# B&R Automation Studio project acopos6d_issues (part 3)

#### brdkSTR.fun
```iecst
FUNCTION brdkStrAppendUdintToA : DINT (*Appends an UDINT to the end of a string. $RETURN=length;Length of the string.*) (*$GROUP=User,$CAT=User,$GROUPICON=User.png,$CATICON=User.png*)
	VAR_INPUT
		value : UDINT; (*UDINT value to be converted.*)
		pString : UDINT; (*String pointer to source string.*)
		base : USINT; (*0,10 = decimal, 2 = binary, 16 = hex.*)
		position : DINT; (*Append position. Negative numbers will count from end of string.*)
	END_VAR
END_FUNCTION

FUNCTION brdkStrAToDint : DINT (*Converts a string to a DINT type. $RETURN=value;DINT value.*) (*$GROUP=User,$CAT=User,$GROUPICON=User.png,$CATICON=User.png*)
	VAR_INPUT
		pString : UDINT; (*String pointer to source string.*)
		base : USINT; (*0,10 = decimal, 2 = binary, 16 = hex.*)
	END_VAR
END_FUNCTION

FUNCTION brdkStrAToDTStructure : DINT (*Converts a STRING of format yyyy-mm-dd hh:mm:ss.ms into a DTStructure. $RETURN=length;Length of the string.*) (*$GROUP=User,$CAT=User,$GROUPICON=User.png,$CATICON=User.png*)
	VAR_INPUT
		pString : UDINT; (*String pointer to source string.*)
		pDTStructure : UDINT; (*Pointer to the DTStructure.*)
	END_VAR
END_FUNCTION

FUNCTION brdkStrAToUdint : UDINT (*Converts a string to an UDINT type. $RETURN=value;UDINT value.*) (*$GROUP=User,$CAT=User,$GROUPICON=User.png,$CATICON=User.png*)
	VAR_INPUT
		pString : UDINT; (*String pointer to source string.*)
		base : USINT; (*0,10 = decimal, 2 = binary, 16 = hex.*)
	END_VAR
END_FUNCTION

FUNCTION brdkStrCat : UDINT (*Appends a copy of the source string to the end of the destination string. $RETURN=address;Address after the string.*) (*$GROUP=User,$CAT=User,$GROUPICON=User.png,$CATICON=User.png*)
	VAR_INPUT
		pDestination : UDINT; (*Destination string pointer.*)
		pSource : UDINT; (*Source string pointer.*)
	END_VAR
END_FUNCTION

FUNCTION brdkStrCatAtChar : DINT (*Appends a copy of the source string to the char position of the destination string. $RETURN=index;Index in destination string where the source string is appended. -1 if char is not found.*) (*$GROUP=User,$CAT=User,$GROUPICON=User.png,$CATICON=User.png*)
	VAR_INPUT
		pDestination : UDINT; (*Destination string pointer.*)
		pSource : UDINT; (*Source string pointer.*)
		pChar : UDINT; (*Char pointer.*)
		direction : DINT; (*0 = first appearance of char, -1 = last appearance of char.*)
		greedy : BOOL; (*If true the source string is appended to the char position. If false the char is still present in the destination string.*)
	END_VAR
END_FUNCTION

FUNCTION brdkStrCharAt : USINT (*Returns the character at the specified index. $RETURN=coding;ASCII coding of the char.*) (*$GROUP=User,$CAT=User,$GROUPICON=User.png,$CATICON=User.png*)
	VAR_INPUT
		pString : UDINT; (*String pointer to source string.*)
		index : UDINT; (*Look up index.*)
		pChar : UDINT; (*Char pointer to char to look up.*)
	END_VAR
END_FUNCTION

FUNCTION brdkStrCharCount : DINT (*Finds how many times a character appears in a string. $RETURN=count;Char count. -1 if error.*) (*$GROUP=User,$CAT=User,$GROUPICON=User.png,$CATICON=User.png*)
	VAR_INPUT
		pString : UDINT; (*String pointer to source string.*)
		pChar : UDINT; (*Pointer to search char.*)
	END_VAR
END_FUNCTION

FUNCTION brdkStrCmp : DINT (*Compares character(s) from string1 to string2. $RETURN=result;0 means that the two string are equal.*)
	VAR_INPUT
		pString1 : UDINT; (*String1 pointer.*)
		pString2 : UDINT; (*String2 pointer.*)
	END_VAR
END_FUNCTION

FUNCTION brdkStrCpy : UDINT (*Copies a string to another string. $RETURN=address;Address after the string.*) (*$GROUP=User,$CAT=User,$GROUPICON=User.png,$CATICON=User.png*)
	VAR_INPUT
		pDestination : UDINT; (*Destination string pointer.*)
		pSource : UDINT; (*Source string pointer.*)
	END_VAR
END_FUNCTION

FUNCTION brdkStrCrc32 : UDINT (*Calculates a CRC32 checksum based on the input string. $RETURN=checksum;Checksum of the string.*) (*$GROUP=User,$CAT=User,$GROUPICON=User.png,$CATICON=User.png*)
	VAR_INPUT
		pString : UDINT; (*String pointer.*)
	END_VAR
END_FUNCTION

FUNCTION brdkStrDintToA : DINT (*Converts a DINT into a STRING type. $RETURN=length;Length of the string.*) (*$GROUP=User,$CAT=User,$GROUPICON=User.png,$CATICON=User.png*)
	VAR_INPUT
		value : DINT; (*DINT value to be converted.*)
		pString : UDINT; (*String pointer to source string.*)
		base : USINT; (*0,10 = decimal, 2 = binary, 16 = hex.*)
	END_VAR
END_FUNCTION

FUNCTION brdkStrDTStructureToA : DINT (*Converts a DTStructure into a STRING type in format yyyy-mm-dd hh:mm:ss.ms. $RETURN=length;Length of the string.*) (*$GROUP=User,$CAT=User,$GROUPICON=User.png,$CATICON=User.png*)
	VAR_INPUT
		pDTStructure : UDINT; (*Pointer to the DTStructure.*)
		pString : UDINT; (*String pointer to destination string.*)
	END_VAR
END_FUNCTION

FUNCTION brdkStrEncode : DINT (*Encodes a string into different formats. $RETURN=address;Address after the string.*) (*$GROUP=User,$CAT=User,$GROUPICON=User.png,$CATICON=User.png*)
	VAR_INPUT
		pDestination : UDINT; (*Destination string pointer.*)
		pSource : UDINT; (*Source string pointer.*)
		format : USINT; (*0 = UTF-8*)
	END_VAR
END_FUNCTION

FUNCTION brdkStrFill : DINT (*Inserts amount of character(s) to the specified position of the string. $RETURN=length;Length of the string. -1 if error.*) (*$GROUP=User,$CAT=User,$GROUPICON=User.png,$CATICON=User.png*)
	VAR_INPUT
		pString : UDINT; (*String pointer to source string.*)
		amount : DINT; (*Fill char amount.*)
		pChar : UDINT; (*Fill char. If 0 whitespace is used.*)
		position : DINT; (*Fill position. Negative numbers will count from end of string.*)
	END_VAR
END_FUNCTION

FUNCTION brdkStrFillUp : DINT (*Fills x amount of character(s) to the specified position of the string. $RETURN=amount;Amount of chars filled. -1 if error.*) (*$GROUP=User,$CAT=User,$GROUPICON=User.png,$CATICON=User.png*)
	VAR_INPUT
		pString : UDINT; (*String pointer to source string.*)
		maxLength : DINT; (*Maximum length of the string.*)
		pChar : UDINT; (*Fill char. If 0 whitespace is used.*)
		position : DINT; (*Fill position. Negative numbers will count from end of string.*)
	END_VAR
END_FUNCTION

FUNCTION brdkStrIndexOf : DINT (*Returns the index within this string of the first or last occurrence of the specified character. $RETURN=index;Index of the char. -1 if char is not found.*) (*$GROUP=User,$CAT=User,$GROUPICON=User.png,$CATICON=User.png*)
	VAR_INPUT
		pString : UDINT; (*String pointer to source string.*)
		pChar : UDINT; (*Char pointer to char to look up.*)
		direction : DINT; (*0 = search from left, -1 = search from right.*)
	END_VAR
END_FUNCTION

FUNCTION brdkStrInsertAtPos : DINT (*Inserts a string into another string at a specified position. $RETURN=length;Length of the string. -1 if error.*) (*$GROUP=User,$CAT=User,$GROUPICON=User.png,$CATICON=User.png*)
	VAR_INPUT
		pString : UDINT; (*String pointer to source string.*)
		pInsert : UDINT; (*String pointer to insert string.*)
		position : DINT; (*Insert position. Negative numbers will count from end of string.*)
	END_VAR
END_FUNCTION

FUNCTION brdkStrIsAlphabet : BOOL (*Returns false or true depending of all characters are present in the alphabet. $RETURN=false/true; a..z = true.*) (*$GROUP=User,$CAT=User,$GROUPICON=User.png,$CATICON=User.png*)
	VAR_INPUT
		pString : UDINT; (*String pointer.*)
	END_VAR
END_FUNCTION

FUNCTION brdkStrIsDigit : BOOL (*Returns false or true depending of all characters are digits. $RETURN=false/true; 0..9 = true.*) (*$GROUP=User,$CAT=User,$GROUPICON=User.png,$CATICON=User.png*)
	VAR_INPUT
		pString : UDINT; (*String pointer.*)
	END_VAR
END_FUNCTION

FUNCTION brdkStrIsEmpty : BOOL (*Returns false or true depending of characters are present in the first position of the string. $RETURN=false/true;Position [0] = /0 = false. Position [0] != /0 = true.*) (*$GROUP=User,$CAT=User,$GROUPICON=User.png,$CATICON=User.png*)
	VAR_INPUT
		pString : UDINT; (*String pointer.*)
	END_VAR
END_FUNCTION

FUNCTION brdkStrJoin : DINT (*Joins elements from a string array into a string with a delimiter. $RETURN=length;Length of the string or error codes.*) (*$GROUP=User,$CAT=User,$GROUPICON=User.png,$CATICON=User.png*)
	VAR_INPUT
		pString : UDINT; (*String pointer to destination string.*)
		pArray : UDINT; (*Pointer to source string array.*)
		pDelimiter : UDINT; (*Delimiter char. If 0 whitespace is used. The delimiter can only be 1 char long.*)
		sizeOfArray : UDINT; (*Max. size of the string array. Size means number of elements in array.*)
		sizeOfArrayString : UDINT; (*Max. size of strings in the array.*)
		sizeOfString : UDINT; (*Max. size of destination string.*)
	END_VAR
END_FUNCTION

FUNCTION brdkStrLen : DINT (*Returns the number of characters in a string. Stops at \0. $RETURN=length;length of the string*) (*$GROUP=User,$CAT=User,$GROUPICON=User.png,$CATICON=User.png*)
	VAR_INPUT
		pString : UDINT; (*String pointer.*)
	END_VAR
END_FUNCTION

FUNCTION brdkStrMemClear : UDINT (*Fills amount of 0 to destination. $RETURN=address;Address after the destination.*) (*$GROUP=User,$CAT=User,$GROUPICON=User.png,$CATICON=User.png*)
	VAR_INPUT
		pDestination : UDINT; (*Destination pointer.*)
		amount : UDINT; (*Amount of character(s) to be initialized.*)
	END_VAR
END_FUNCTION

FUNCTION brdkStrMemCmp : DINT (*Compares amount of character(s) from area1 to area2. $RETURN=result;0 means that the two areas are equal.*) (*$GROUP=User,$CAT=User,$GROUPICON=User.png,$CATICON=User.png*)
	VAR_INPUT
		pArea1 : UDINT; (*Area1 pointer.*)
		pArea2 : UDINT; (*Area2 pointer.*)
		amount : UDINT; (*Amount of character(s) to be comared.*)
	END_VAR
END_FUNCTION

FUNCTION brdkStrMemCpy : UDINT (*Copies amount of character(s) from source to destination. $RETURN=address;Address after the destination.*) (*$GROUP=User,$CAT=User,$GROUPICON=User.png,$CATICON=User.png*)
	VAR_INPUT
		pDestination : UDINT; (*Destination pointer.*)
		pSource : UDINT; (*Source pointer.*)
		amount : UDINT; (*Amount of character(s) to be copied.*)
	END_VAR
END_FUNCTION

FUNCTION brdkStrMemMove : UDINT (*Moves amount of character(s) from source to destination. $RETURN=address;Address after the destination.*) (*$GROUP=User,$CAT=User,$GROUPICON=User.png,$CATICON=User.png*)
	VAR_INPUT
		pDestination : UDINT; (*Destination pointer.*)
		pSource : UDINT; (*Source pointer.*)
		amount : UDINT; (*Amount of character(s) to be moved.*)
	END_VAR
END_FUNCTION

FUNCTION brdkStrMemSet : UDINT (*Fills amount of character(s) to destination. $RETURN=address;Address after the destination.*) (*$GROUP=User,$CAT=User,$GROUPICON=User.png,$CATICON=User.png*)
	VAR_INPUT
		pDestination : UDINT; (*Destination pointer.*)
		value : USINT; (*Initialization value.*)
		amount : UDINT; (*Amount of character(s) to be initialized.*)
	END_VAR
END_FUNCTION

FUNCTION brdkStrMove : UDINT (*Moves a string to another string. $RETURN=address;Address after the string.*) (*$GROUP=User,$CAT=User,$GROUPICON=User.png,$CATICON=User.png*)
	VAR_INPUT
		pDestination : UDINT; (*Destination string pointer.*)
		pSource : UDINT; (*Source string pointer.*)
	END_VAR
END_FUNCTION

FUNCTION brdkStrNAToDint : DINT (*Converts a string to an DINT type for amount of characters. If the function encounters a null character in the source string, if will stop. $RETURN=value;DINT value.*) (*$GROUP=User,$CAT=User,$GROUPICON=User.png,$CATICON=User.png*)
	VAR_INPUT
		pString : UDINT; (*String pointer to source string.*)
		amount : UDINT; (*Amount of character(s) to be converted.*)
		base : USINT; (*0,10 = decimal, 2 = binary, 16 = hex.*)
	END_VAR
END_FUNCTION

FUNCTION brdkStrNAToUdint : UDINT (*Converts a string to an UDINT type for amount of characters. If the function encounters a null character in the source string, if will stop. $RETURN=value;UDINT value.*) (*$GROUP=User,$CAT=User,$GROUPICON=User.png,$CATICON=User.png*)
	VAR_INPUT
		pString : UDINT; (*String pointer to source string.*)
		amount : UDINT; (*Amount of character(s) to be converted.*)
		base : USINT; (*0,10 = decimal, 2 = binary, 16 = hex.*)
	END_VAR
END_FUNCTION

FUNCTION brdkStrNCpy : UDINT (*Copies a string to another string. If the function encounters a null character in the source string, the function will add null characters to the destination string until amount character(s) have been written. $RETURN=address;Address after the string.*) (*$GROUP=User,$CAT=User,$GROUPICON=User.png,$CATICON=User.png*)
	VAR_INPUT
		pDestination : UDINT; (*Destination string pointer.*)
		pSource : UDINT; (*Source string pointer.*)
		amount : UDINT; (*Amount of character(s) to be moved.*)
	END_VAR
END_FUNCTION

FUNCTION brdkStrNIsAlphabet : BOOL (*Returns false or true depending of the amount of characters are present in the alphabet. $RETURN=false/true; a..z = true.*) (*$GROUP=User,$CAT=User,$GROUPICON=User.png,$CATICON=User.png*)
	VAR_INPUT
		pString : UDINT; (*String pointer.*)
		amount : UDINT; (*Amount of character(s) to be checked.*)
	END_VAR
END_FUNCTION

FUNCTION brdkStrNIsDigit : BOOL (*Returns false or true depending of the amount characters are digits. $RETURN=false/true; 0..9 = true.*) (*$GROUP=User,$CAT=User,$GROUPICON=User.png,$CATICON=User.png*)
	VAR_INPUT
		pString : UDINT; (*String pointer.*)
		amount : UDINT; (*Amount of character(s) to be checked.*)
	END_VAR
END_FUNCTION

FUNCTION brdkStrRemove : UDINT (*Removes character(s) from a string from a specified position. $RETURN=address;Address after the string.*) (*$GROUP=User,$CAT=User,$GROUPICON=User.png,$CATICON=User.png*)
	VAR_INPUT
		pString : UDINT; (*Source string pointer.*)
		start : DINT; (*Index of where to start in the string. Negative numbers start from the end of the string.*)
		length : DINT; (*0 means to the end of the string. Negative length is subtracted from the end of the string. Is start is negative length is subtracted from the start of the string. *)
	END_VAR
END_FUNCTION

FUNCTION brdkStrRepeat : DINT (*Repeats a string a specified number of times. $RETURN=length;Length of the string.*) (*$GROUP=User,$CAT=User,$GROUPICON=User.png,$CATICON=User.png*)
	VAR_INPUT
		pString : UDINT; (*String pointer to source string.*)
		times : DINT; (*Number of times the string should be repeated.*)
	END_VAR
END_FUNCTION

FUNCTION brdkStrReplace : DINT (*Replaces some characters with some other characters in a string. $RETURN=number;Number of replacements done.*) (*$GROUP=User,$CAT=User,$GROUPICON=User.png,$CATICON=User.png*)
	VAR_INPUT
		pString : UDINT; (*String pointer to source string.*)
		pFind : UDINT; (*String pointer to find string.*)
		pReplace : UDINT; (*String pointer to replacement string:*)
	END_VAR
END_FUNCTION

FUNCTION brdkStrReverse : DINT (*Reverses a string from start position to end position. $RETURN=count;Number of reverses done. -1 if error.*) (*$GROUP=User,$CAT=User,$GROUPICON=User.png,$CATICON=User.png*)
	VAR_INPUT
		pString : UDINT; (*String pointer to source string.*)
		startPosition : DINT; (*Start position. Must be a positive number and less than length.*)
		endPosition : DINT; (*End position. Must be less than length unless it's a negative numbers which will count from end of string.*)
	END_VAR
END_FUNCTION

FUNCTION brdkStrReverseWords : DINT (*Reverses words in a string. $RETURN=count;Number of words reversed.*) (*$GROUP=User,$CAT=User,$GROUPICON=User.png,$CATICON=User.png*)
	VAR_INPUT
		pString : UDINT; (*String pointer to source string.*)
	END_VAR
END_FUNCTION

FUNCTION brdkStrSearch : DINT (*Searches a string for a specified string. $RETURN=position; Position of the match. -1 if no match.*) (*$GROUP=User,$CAT=User,$GROUPICON=User.png,$CATICON=User.png*)
	VAR_INPUT
		pString : UDINT; (*String pointer to source string.*)
		pSearchString : UDINT; (*String pointer to search string.*)
	END_VAR
END_FUNCTION

FUNCTION brdkStrSlice : DINT (*Slices a part of a string. $RETURN=length;Length of the string. -1 if error.*) (*$GROUP=User,$CAT=User,$GROUPICON=User.png,$CATICON=User.png*)
	VAR_INPUT
		pString : UDINT; (*String pointer to source string.*)
		start : DINT; (*Start position.*)
		end : DINT; (*End position.*)
	END_VAR
END_FUNCTION

FUNCTION brdkStrSplit : DINT (*Splits a string into an array of string using a seperator. $RETURN=count;Number of elements splitted or an error code.*) (*$GROUP=User,$CAT=User,$GROUPICON=User.png,$CATICON=User.png*)
	VAR_INPUT
		pArray : UDINT; (*Pointer to destination string array.*)
		pString : UDINT; (*String pointer to source string.*)
		pDelimiter : UDINT; (*Delimiter char. If 0 whitespace is used. The delimiter can only be 1 char long.*)
		sizeOfArray : UDINT; (*Max. size of the string array. Size means number of elements in array.*)
		sizeofArrayString : UDINT; (*Max. size of strings in the array.*)
		greedy : BOOL; (*Remove or keep the seperator from the string.*)
	END_VAR
END_FUNCTION

FUNCTION brdkStrSubDintSearch : DINT (*Returns a DINT based on a search. $RETURN=length;Length of the destination string. -1 if error.*) (*$GROUP=User,$CAT=User,$GROUPICON=User.png,$CATICON=User.png*)
	VAR_INPUT
		pSource : UDINT; (*Source string pointer.*)
		pStart : UDINT; (*String pointer for start search string.*)
		pEnd : UDINT; (*String pointer for end search string. The function will only search after the start string.*)
		startOffset : DINT; (*Offset for the start poition. If greedy = true offset is after the start has been removed.*)
		base : USINT; (*0,10 = decimal, 2 = binary, 16 = hex.*)
	END_VAR
END_FUNCTION

FUNCTION brdkStrSubStr : DINT (*Returns a part of a string. $RETURN=length;Length of the destination string. -1 if error.*) (*$GROUP=User,$CAT=User,$GROUPICON=User.png,$CATICON=User.png*)
	VAR_INPUT
		pDestination : UDINT; (*Destination string pointer.*)
		pSource : UDINT; (*Source string pointer.*)
		start : DINT; (*Index of where to start in the string. Negative numbers start from the end of the string.*)
		length : DINT; (*0 means to the end of the string. Negative length is subtracted from the end of the string. Is start is negative length is subtracted from the start of the string. *)
	END_VAR
END_FUNCTION

FUNCTION brdkStrSubStrSearch : BOOL (*Returns a part of a string based on a search. $RETURN=success;TRUE = success *) (*$GROUP=User,$CAT=User,$GROUPICON=User.png,$CATICON=User.png*)
	VAR_INPUT
		pDestination : UDINT; (*Destination string pointer.*)
		pSource : UDINT; (*Source string pointer.*)
		pStart : UDINT; (*String pointer for start search string.*)
		pEnd : UDINT; (*String pointer for end search string. The function will only search after the start string.*)
		startOffset : DINT; (*Offset for the start poition. If greedy = true offset is after the start has been removed.*)
		greedy : BOOL; (*Will add or remove the search strings from the destination string.*)
	END_VAR
END_FUNCTION

FUNCTION brdkStrToDec : DINT (*Converts a string of hexadecimal values to ASCII characters. $RETURN=length;Length of the string. -1 if error.*) (*$GROUP=User,$CAT=User,$GROUPICON=User.png,$CATICON=User.png*)
	VAR_INPUT
		pString : UDINT; (*String pointer to source string.*)
	END_VAR
END_FUNCTION

FUNCTION brdkStrToHex : DINT (*Converts a string of ASCII characters to hexadecimal values. $RETURN=length;Length of the string.*) (*$GROUP=User,$CAT=User,$GROUPICON=User.png,$CATICON=User.png*)
	VAR_INPUT
		pString : UDINT; (*String pointer to source string.*)
	END_VAR
END_FUNCTION

FUNCTION brdkStrToLowerCase : DINT (*Converts a string to lowercase letters. $RETURN=number;Number of characters changed.*) (*$GROUP=User,$CAT=User,$GROUPICON=User.png,$CATICON=User.png*)
	VAR_INPUT
		pString : UDINT; (*String pointer to source string.*)
	END_VAR
END_FUNCTION

FUNCTION brdkStrToUpperCase : DINT (*Converts a string to uppercase letters. $RETURN=number;Number of characters changed.*) (*$GROUP=User,$CAT=User,$GROUPICON=User.png,$CATICON=User.png*)
	VAR_INPUT
		pString : UDINT; (*String pointer to source string.*)
	END_VAR
END_FUNCTION

FUNCTION brdkStrToUpperCaseWords : DINT (*Convert the first character of each word to uppercase. (title()). $RETURN=number;Number of characters changed.*) (*$GROUP=User,$CAT=User,$GROUPICON=User.png,$CATICON=User.png*)
	VAR_INPUT
		pString : UDINT; (*String pointer to source string.*)
	END_VAR
END_FUNCTION

FUNCTION brdkStrTrim : DINT (*Removes whitespaces from a string. $RETURN=number;Number of whitespaces removed from string.*) (*$GROUP=User,$CAT=User,$GROUPICON=User.png,$CATICON=User.png*)
	VAR_INPUT
		pString : UDINT; (*String pointer to source string.*)
		direction : DINT; (*0 = both sides, 1 = left side only, -1 = right side only.*)
	END_VAR
END_FUNCTION

FUNCTION brdkStrUdintToA : DINT (*Converts an UDINT into a STRING type. $RETURN=length;Length of the string.*) (*$GROUP=User,$CAT=User,$GROUPICON=User.png,$CATICON=User.png*)
	VAR_INPUT
		value : UDINT; (*UDINT value to be converted.*)
		pString : UDINT; (*String pointer to source string.*)
		base : USINT; (*0,10 = decimal, 2 = binary, 16 = hex.*)
	END_VAR
END_FUNCTION

FUNCTION brdkStrWord : DINT (*Returns a word in a string given by a number and a delimiter. $RETURN=length;Length of the string.*) (*$GROUP=User,$CAT=User,$GROUPICON=User.png,$CATICON=User.png*)
	VAR_INPUT
		pDestination : UDINT; (*Destination string pointer.*)
		pSource : UDINT; (*Source string pointer.*)
		pDelimiter : UDINT; (*Delimiter char. If 0 whitespace is used. The delimiter can only be 1 char long.*)
		number : DINT; (*Word number in string. 1 = first word. -1 = last word.*)
		sizeOfString : UDINT; (*Max. size of destination string.*)
	END_VAR
END_FUNCTION
```

#### brdkSTR.var
```iecst
VAR CONSTANT
	BRDK_STR_RIGHT_TRIM : DINT := -1; (*trims right side only*)
	BRDK_STR_LEFT_TRIM : DINT := 1; (*trims left side only*)
	BRDK_STR_CONVERT_HEX : USINT := 16; (*converts to/from hex*)
	BRDK_STR_CONVERT_DECIMAL : USINT := 10; (*converts to/from decimal*)
	BRDK_STR_CONVERT_BINARY : USINT := 2; (*converts to/from binary*)
	BRDK_STR_BOTH_TRIM : DINT := 0; (*trims both sides*)
	BRDK_STR_RIGHT_SEARCH : DINT := -1; (*search from right side*)
	BRDK_STR_LEFT_SEARCH : DINT := 0; (*search from left side*)
	BRDK_STR_UTF_8 : USINT := 0; (*encoding in utf-8 format*)
END_VAR
(*ASCII CONTROL CHARACTERS 0 - 31*)
VAR CONSTANT
	BRDK_STR_ASCII_NULL : USINT := 0; (*null*)
	BRDK_STR_ASCII_SOH : USINT := 1; (*start of heading*)
	BRDK_STR_ASCII_STX : USINT := 2; (*start of text*)
	BRDK_STR_ASCII_ETX : USINT := 3; (*end of text*)
	BRDK_STR_ASCII_EOT : USINT := 4; (*end of transmission*)
	BRDK_STR_ASCII_ENQ : USINT := 5; (*enquiry*)
	BRDK_STR_ASCII_ACK : USINT := 6; (*acknowledge*)
	BRDK_STR_ASCII_BEL : USINT := 7; (*bell*)
	BRDK_STR_ASCII_BS : USINT := 8; (*backspace*)
	BRDK_STR_ASCII_TAB : USINT := 9; (*horizontal tab*)
	BRDK_STR_ASCII_LF : USINT := 10; (*line feed*)
	BRDK_STR_ASCII_VT : USINT := 11; (*vertical tab*)
	BRDK_STR_ASCII_FF : USINT := 12; (*NP form feed, new page*)
	BRDK_STR_ASCII_CR : USINT := 13; (*carriage return*)
	BRDK_STR_ASCII_SO : USINT := 14; (*shift out*)
	BRDK_STR_ASCII_SI : USINT := 15; (*shift in*)
	BRDK_STR_ASCII_DLE : USINT := 16; (*data link escape*)
	BRDK_STR_ASCII_DC1 : USINT := 17; (*device control 1*)
	BRDK_STR_ASCII_DC2 : USINT := 18; (*device control 2*)
	BRDK_STR_ASCII_DC3 : USINT := 19; (*device control 3*)
	BRDK_STR_ASCII_DC4 : USINT := 20; (*device control 4*)
	BRDK_STR_ASCII_NAK : USINT := 21; (*negative acknowledge*)
	BRDK_STR_ASCII_SYN : USINT := 22; (*synchronous idle*)
	BRDK_STR_ASCII_ETB : USINT := 23; (*end of trans. block*)
	BRDK_STR_ASCII_CAN : USINT := 24; (*cancel*)
	BRDK_STR_ASCII_EM : USINT := 25; (*end of medium*)
	BRDK_STR_ASCII_SUB : USINT := 26; (*substitute*)
	BRDK_STR_ASCII_ESC : USINT := 27; (*escape*)
	BRDK_STR_ASCII_FS : USINT := 28; (*file separator*)
	BRDK_STR_ASCII_GS : USINT := 29; (*group separator*)
	BRDK_STR_ASCII_RS : USINT := 30; (*record separator*)
	BRDK_STR_ASCII_US : USINT := 31; (*unit separator*)
END_VAR
(*ASCII PRINTABLE CHARACTERS 32 - 127*)
VAR CONSTANT
	BRDK_STR_ASCII_SPACE : USINT := 32; (*space*)
	BRDK_STR_ASCII_EXCLAMATION : USINT := 33; (*!*)
	BRDK_STR_ASCII_DOUBLE_QUOTES : USINT := 34; (*"*)
	BRDK_STR_ASCII_NUMBER : USINT := 35; (*#*)
	BRDK_STR_ASCII_DOLLAR : USINT := 36; (*$*)
	BRDK_STR_ASCII_PERCENT : USINT := 37; (*%*)
	BRDK_STR_ASCII_AMPERSAND : USINT := 38; (*&*)
	BRDK_STR_ASCII_SINGLE_QUOTE : USINT := 39; (*'*)
	BRDK_STR_ASCII_OPEN_PARENTHESIS : USINT := 40; (*(*)
	BRDK_STR_ASCII_CLOSE_PARENTHESIS : USINT := 41; (*)*)
	BRDK_STR_ASCII_ASTERIX : USINT := 42; (***)
	BRDK_STR_ASCII_PLUS : USINT := 43; (*+*)
	BRDK_STR_ASCII_COMMA : USINT := 44; (*,*)
	BRDK_STR_ASCII_HYPHEN : USINT := 45; (*-*)
	BRDK_STR_ASCII_DOT : USINT := 46; (*.*)
	BRDK_STR_ASCII_FRONT_SLASH : USINT := 47; (*/*)
	BRDK_STR_ASCII_0 : USINT := 48; (*0*)
	BRDK_STR_ASCII_1 : USINT := 49; (*1*)
	BRDK_STR_ASCII_2 : USINT := 50; (*2*)
	BRDK_STR_ASCII_3 : USINT := 51; (*3*)
	BRDK_STR_ASCII_4 : USINT := 52; (*4*)
	BRDK_STR_ASCII_5 : USINT := 53; (*5*)
	BRDK_STR_ASCII_6 : USINT := 54; (*6*)
	BRDK_STR_ASCII_7 : USINT := 55; (*7*)
	BRDK_STR_ASCII_8 : USINT := 56; (*8*)
	BRDK_STR_ASCII_9 : USINT := 57; (*9*)
	BRDK_STR_ASCII_COLON : USINT := 58; (*:*)
	BRDK_STR_ASCII_SEMI_COLON : USINT := 59; (*;*)
	BRDK_STR_ASCII_LESS_THAN : USINT := 60; (*<*)
	BRDK_STR_ASCII_EQUALS : USINT := 61; (*=*)
	BRDK_STR_ASCII_GREATER_THAN : USINT := 62; (*>*)
	BRDK_STR_ASCII_QUESTION : USINT := 63; (*?*)
	BRDK_STR_ASCII_AT : USINT := 64; (*@*)
	BRDK_STR_ASCII_A : USINT := 65; (*A*)
	BRDK_STR_ASCII_B : USINT := 66; (*B*)
	BRDK_STR_ASCII_C : USINT := 67; (*C*)
	BRDK_STR_ASCII_D : USINT := 68; (*D*)
	BRDK_STR_ASCII_E : USINT := 69; (*E*)
	BRDK_STR_ASCII_F : USINT := 70; (*F*)
	BRDK_STR_ASCII_G : USINT := 71; (*G*)
	BRDK_STR_ASCII_H : USINT := 72; (*H*)
	BRDK_STR_ASCII_I : USINT := 73; (*I*)
	BRDK_STR_ASCII_J : USINT := 74; (*J*)
	BRDK_STR_ASCII_K : USINT := 75; (*K*)
	BRDK_STR_ASCII_L : USINT := 76; (*L*)
	BRDK_STR_ASCII_M : USINT := 77; (*M*)
	BRDK_STR_ASCII_N : USINT := 78; (*N*)
	BRDK_STR_ASCII_O : USINT := 79; (*O*)
	BRDK_STR_ASCII_P : USINT := 80; (*P*)
	BRDK_STR_ASCII_Q : USINT := 81; (*Q*)
	BRDK_STR_ASCII_R : USINT := 82; (*R*)
	BRDK_STR_ASCII_S : USINT := 83; (*S*)
	BRDK_STR_ASCII_T : USINT := 84; (*T*)
	BRDK_STR_ASCII_U : USINT := 85; (*U*)
	BRDK_STR_ASCII_V : USINT := 86; (*V*)
	BRDK_STR_ASCII_W : USINT := 87; (*W*)
	BRDK_STR_ASCII_X : USINT := 88; (*X*)
	BRDK_STR_ASCII_Y : USINT := 89; (*Y*)
	BRDK_STR_ASCII_Z : USINT := 90; (*Z*)
	BRDK_STR_ASCII_OPEN_BRACKET : USINT := 91; (*[*)
	BRDK_STR_ASCII_BACK_SLASH : USINT := 92; (*\*)
	BRDK_STR_ASCII_CLOSE_BRACKET : USINT := 93; (*]*)
	BRDK_STR_ASCII_CARET : USINT := 94; (*^*)
	BRDK_STR_ASCII_UNDERSCORE : USINT := 95; (*_*)
	BRDK_STR_ASCII_GRAVE_ACCENT : USINT := 96; (*`*)
	BRDK_STR_ASCII_a : USINT := 97; (*a*)
	BRDK_STR_ASCII_b : USINT := 98; (*b*)
	BRDK_STR_ASCII_c : USINT := 99; (*c*)
	BRDK_STR_ASCII_d : USINT := 100; (*d*)
	BRDK_STR_ASCII_e : USINT := 101; (*e*)
	BRDK_STR_ASCII_f : USINT := 102; (*f*)
	BRDK_STR_ASCII_g : USINT := 103; (*g*)
	BRDK_STR_ASCII_h : USINT := 104; (*h*)
	BRDK_STR_ASCII_i : USINT := 105; (*i*)
	BRDK_STR_ASCII_j : USINT := 106; (*j*)
	BRDK_STR_ASCII_k : USINT := 107; (*k*)
	BRDK_STR_ASCII_l : USINT := 108; (*l*)
	BRDK_STR_ASCII_m : USINT := 109; (*m*)
	BRDK_STR_ASCII_n : USINT := 110; (*n*)
	BRDK_STR_ASCII_o : USINT := 111; (*o*)
	BRDK_STR_ASCII_p : USINT := 112; (*p*)
	BRDK_STR_ASCII_q : USINT := 113; (*q*)
	BRDK_STR_ASCII_r : USINT := 114; (*r*)
	BRDK_STR_ASCII_s : USINT := 115; (*s*)
	BRDK_STR_ASCII_t : USINT := 116; (*t*)
	BRDK_STR_ASCII_u : USINT := 117; (*u*)
	BRDK_STR_ASCII_v : USINT := 118; (*v*)
	BRDK_STR_ASCII_w : USINT := 119; (*w*)
	BRDK_STR_ASCII_x : USINT := 120; (*x*)
	BRDK_STR_ASCII_y : USINT := 121; (*y*)
	BRDK_STR_ASCII_z : USINT := 122; (*z*)
	BRDK_STR_ASCII_OPEN_BRACE : USINT := 123; (*{*)
	BRDK_STR_ASCII_VERTICAL_BAR : USINT := 124; (*|*)
	BRDK_STR_ASCII_CLOSE_BRACE : USINT := 125; (*}*)
	BRDK_STR_ASCII_EQUIVALENCY : USINT := 126; (*~*)
END_VAR
(*ASCII EXTENDED CHARACTERS 128 - 255*)
VAR CONSTANT
	BRDK_STR_ASCII_EURO : USINT := 128; (*€*)
	BRDK_STR_ASCII_SINGLE_LOW_QUOTE : USINT := 130; (*‚*)
	BRDK_STR_ASCII_F_WITH_HOOK : USINT := 131; (*ƒ*)
	BRDK_STR_ASCII_DOUBLE_LOW_QUOTE : USINT := 132; (*„*)
	BRDK_STR_ASCII_HORIZON_ELLIPSIS : USINT := 133; (*…*)
	BRDK_STR_ASCII_DAGGER : USINT := 134; (*†*)
	BRDK_STR_ASCII_DOUBLE_DAGGER : USINT := 135; (*‡*)
	BRDK_STR_ASCII_MOD_CIRCUM_ACCENT : USINT := 136; (*ˆ*)
	BRDK_STR_ASCII_PERMILLE : USINT := 137; (*‰*)
	BRDK_STR_ASCII_S_CAPCON : USINT := 138; (*Š*)
	BRDK_STR_ASCII_LEFT_ANGLE : USINT := 139; (*‹*)
	BRDK_STR_ASCII_OE_SIGN : USINT := 140; (*Œ*)
	BRDK_STR_ASCII_Z_CAPRON : USINT := 142; (*Ž*)
	BRDK_STR_ASCII_LEFT_SINGLE_QUO : USINT := 145; (*‘*)
	BRDK_STR_ASCII_RIGHT_SINGLE_QUO : USINT := 146; (*’*)
	BRDK_STR_ASCII_LEFT_DOUBLE_QUO : USINT := 147; (*“*)
	BRDK_STR_ASCII_RIGHT_DOUBLE_QUO : USINT := 148; (*”*)
	BRDK_STR_ASCII_BULLET : USINT := 149; (*•*)
	BRDK_STR_ASCII_EN_DASH : USINT := 150; (*–*)
	BRDK_STR_ASCII_EM_DASH : USINT := 151; (*—*)
	BRDK_STR_ASCII_SMALL_TILDE : USINT := 152; (*˜*)
	BRDK_STR_ASCII_TRADE_MARK : USINT := 153; (*™*)
	BRDK_STR_ASCII_s_CAPCON : USINT := 154; (*š*)
	BRDK_STR_ASCII_RIGHT_ANGLE : USINT := 155; (*›*)
	BRDK_STR_ASCII_oe : USINT := 156; (*œ*)
	BRDK_STR_ASCII_z_CAPCON : USINT := 158; (*ž*)
END_VAR
```

#### brdkStrAppendUdintToA.c
```c
#include <brdkSTR_func.h>

signed long brdkStrAppendUdintToA(unsigned long value, unsigned long pString, unsigned char base, signed long position) {
	signed long i,cnt=0,len = brdkStrLen(pString);
	signed long start = position > -1 ? position :len+position+1;
	unsigned char tmp;
	i=start;
	tmp = BRDK_STR_ASCII_0;
	base = !base ? 10 : base;	/* make sure base is not 0 */
	if (value != 0) {
		while (value > 0) {
			unsigned long rem = value % base;
			unsigned char tmp = (rem > 9)? (rem-10) + BRDK_STR_ASCII_A : rem + BRDK_STR_ASCII_0;
			brdkStrFill(pString,1,(unsigned long)&tmp,i++);
	       	value = value/base;
			cnt++;
		}
		brdkStrReverse(pString,start,--i);
		return len+cnt;
	}
	else {
		brdkStrFill(pString,1,(unsigned long)&tmp,i);
		return len+1;
	}
}
```

#### brdkStrAToDint.c
```c
#include <brdkSTR_func.h>

signed long brdkStrAToDint(unsigned long pString, unsigned char base) {
	return brdkStrNAToDint(pString, brdkStrLen(pString), base);
}
```

#### brdkStrAToDTStructure.c
```c
#include <brdkSTR_func.h>

signed long brdkStrAToDTStructure(unsigned long pString, unsigned long pDTStructure) {
	/* format must be 2020-01-01 01:01:01,001 */
	DTStructure* dtStruct = (DTStructure*)pDTStructure;
	/* year */
	if(!brdkStrNIsDigit(pString,4)) return -1;
	dtStruct->year = brdkStrNAToUdint(pString, 4, BRDK_STR_CONVERT_DECIMAL);
	if(((char*)pString)[4] != BRDK_STR_ASCII_HYPHEN) return -1;
	/* month */
	if(!brdkStrNIsDigit((unsigned long)&((char*)pString)[5],2)) return -1;
	dtStruct->month = brdkStrNAToUdint((unsigned long)&((char*)pString)[5], 2, BRDK_STR_CONVERT_DECIMAL);
	if(((char*)pString)[7] != BRDK_STR_ASCII_HYPHEN) return -1;
	/* day */
	if(!brdkStrNIsDigit((unsigned long)&((char*)pString)[8],2)) return -1;
	dtStruct->day = brdkStrNAToUdint((unsigned long)&((char*)pString)[8], 2, BRDK_STR_CONVERT_DECIMAL);
	if(((char*)pString)[10] != BRDK_STR_ASCII_SPACE) return -1;
	/* hour */
	if(!brdkStrNIsDigit((unsigned long)&((char*)pString)[11],2)) return -1;
	dtStruct->hour = brdkStrNAToUdint((unsigned long)&((char*)pString)[11], 2, BRDK_STR_CONVERT_DECIMAL);
	if(((char*)pString)[13] != BRDK_STR_ASCII_COLON) return -1;
	/* minute */
	if(!brdkStrNIsDigit((unsigned long)&((char*)pString)[14],2)) return -1;
	dtStruct->minute = brdkStrNAToUdint((unsigned long)&((char*)pString)[14], 2, BRDK_STR_CONVERT_DECIMAL);
	if(((char*)pString)[16] != BRDK_STR_ASCII_COLON) return -1;
	/* second */
	if(!brdkStrNIsDigit((unsigned long)&((char*)pString)[17],2)) return -1;
	dtStruct->second = brdkStrNAToUdint((unsigned long)&((char*)pString)[17], 2, BRDK_STR_CONVERT_DECIMAL);
	if(((char*)pString)[19] != BRDK_STR_ASCII_DOT) return -1;
	/* millisecond */
	if(!brdkStrNIsDigit((unsigned long)&((char*)pString)[20],3)) return -1;
	dtStruct->millisec = brdkStrNAToUdint((unsigned long)&((char*)pString)[20], 3, BRDK_STR_CONVERT_DECIMAL);
	dtStruct->wday = dayOfWeek(dtStruct->day,dtStruct->month,dtStruct->year);
	return 0;
}
```

#### brdkStrAToUdint.c
```c
#include <brdkSTR_func.h>

unsigned long brdkStrAToUdint(unsigned long pString, unsigned char base) {
	return brdkStrNAToUdint(pString, brdkStrLen(pString), base);
}
```

#### brdkStrCat.c
```c
#include <brdkSTR_func.h>

unsigned long brdkStrCat(unsigned long pDestination, unsigned long pSource) {
	unsigned long i=0,len = brdkStrLen(pSource), start = brdkStrLen(pDestination);
	for(i=0; i< len; i++) ((char*)pDestination)[start+i] = ((char*)pSource)[i];
	((char*)pDestination)[start+i] = BRDK_STR_ASCII_NULL;
	return pDestination+start+i;
}
```

#### brdkStrCatAtChar.c
```c
#include <brdkSTR_func.h>

signed long brdkStrCatAtChar(unsigned long pDestination, unsigned long pSource, unsigned long pChar, signed long direction, unsigned char greedy) {
	unsigned long i=0,len = brdkStrLen(pSource);
	signed long start = brdkStrIndexOf(pDestination,pChar,direction);
	if(start > -1) {
		start += !greedy;
		for(i=0; i< len; i++) ((char*)pDestination)[start+i] = ((char*)pSource)[i];
		((char*)pDestination)[start+i] = BRDK_STR_ASCII_NULL;
	}
	return start;
}
```

#### brdkStrCharAt.c
```c
#include <brdkSTR_func.h>

unsigned char brdkStrCharAt(unsigned long pString, unsigned long index, unsigned long pChar) {
	if(index < brdkStrLen(pString)) {
		*(char*)pChar = ((char*)pString)[index];
		return ((char*)pString)[index];
	}
	else {
		*(char*)pChar = BRDK_STR_ASCII_NULL;
		return 0;
	}
}
```

#### brdkStrCharCount.c
```c
#include <brdkSTR_func.h>

signed long brdkStrCharCount(unsigned long pString, unsigned long pChar) {
	signed long i=0, cnt=0;
	if(pChar != 0 && *(char*)pChar != 0) {
		while(((char*)pString)[i]) if(((char*)pString)[i++] == *(char*)pChar) cnt++;
	}
	else cnt = -1;
	return cnt;
}
```

#### brdkStrCmp.c
```c
#include <brdkSTR_func.h>

signed long brdkStrCmp(unsigned long pString1, unsigned long pString2) {
	unsigned long i=0;
	do if(((char*)pString1)[i] != ((char*)pString2)[i]) break;
	while(((char*)pString1)[i] != BRDK_STR_ASCII_NULL && ((char*)pString2)[i++] != BRDK_STR_ASCII_NULL);
	return ((char*)pString1)[i]-((char*)pString2)[i];
}
```

#### brdkStrCpy.c
```c
#include <brdkSTR_func.h>

unsigned long brdkStrCpy(unsigned long pDestination, unsigned long pSource) {
	unsigned long i=0;
	do ((char*)pDestination)[i] = ((char*)pSource)[i];
	while(((char*)pSource)[i++] != BRDK_STR_ASCII_NULL);
	return pDestination+i;
}
```

#### brdkStrCrc32.c
```c
#include <brdkSTR_func.h>

unsigned long brdkStrCrc32(unsigned long pString) {
	int i=0, crc = 0xFFFFFFFF;
	unsigned int byte, c;
	const unsigned int g0 = 0xEDB88320, g1 = g0>>1,g2 = g0>>2, g3 = g0>>3, g4 = g0>>4, g5 = g0>>5, g6 = (g0>>6)^g0, g7 = ((g0>>6)^g0)>>1;
	while ((byte = ((char*)pString)[i]) != BRDK_STR_ASCII_NULL) {    /* Get next byte. */
		crc = crc ^ byte;
		c = ((crc<<31>>31) & g7) ^ ((crc<<30>>31) & g6) ^
			((crc<<29>>31) & g5) ^ ((crc<<28>>31) & g4) ^
			((crc<<27>>31) & g3) ^ ((crc<<26>>31) & g2) ^
			((crc<<25>>31) & g1) ^ ((crc<<24>>31) & g0);
		crc = ((unsigned)crc >> 8) ^ c;
		i++;
   }
   return ~crc;
}
```

#### brdkStrDintToA.c
```c
#include <brdkSTR_func.h>

signed long brdkStrDintToA(signed long value, unsigned long pString, unsigned char base) {
	if(value < 0) {
		((char*)pString)[0] = BRDK_STR_ASCII_HYPHEN;
		return brdkStrUdintToA(-value,pString+1,BRDK_STR_CONVERT_DECIMAL)+1;
	}
	else return brdkStrUdintToA(value,pString,base);
}
```

#### brdkStrDTStructureToA.c
```c
#include <brdkSTR_func.h>

signed long brdkStrDTStructureToA(unsigned long pDTStructure, unsigned long pString) {
	/* format will be 2020-01-01 01:01:01,001 */
	DTStructure* dtStruct = (DTStructure*)pDTStructure;
	brdkStrUdintToA(dtStruct->year,(unsigned long)&(((char*)pString)[0]),BRDK_STR_CONVERT_DECIMAL);
	((char*)pString)[4] = BRDK_STR_ASCII_HYPHEN;
	if(dtStruct->month < 10) {
		((char*)pString)[5] = BRDK_STR_ASCII_0;
		brdkStrUdintToA(dtStruct->month,(unsigned long)&(((char*)pString)[6]),BRDK_STR_CONVERT_DECIMAL);
	}
	else brdkStrUdintToA(dtStruct->month,(unsigned long)&(((char*)pString)[5]),BRDK_STR_CONVERT_DECIMAL);
	((char*)pString)[7] = BRDK_STR_ASCII_HYPHEN;
	if(dtStruct->day < 10) {
		((char*)pString)[8] = BRDK_STR_ASCII_0;
		brdkStrUdintToA(dtStruct->day,(unsigned long)&(((char*)pString)[9]),BRDK_STR_CONVERT_DECIMAL);
	}
	else brdkStrUdintToA(dtStruct->day,(unsigned long)&(((char*)pString)[8]),BRDK_STR_CONVERT_DECIMAL);
	((char*)pString)[10] = BRDK_STR_ASCII_SPACE;
	if(dtStruct->hour < 10) {
		((char*)pString)[11] = BRDK_STR_ASCII_0;
		brdkStrUdintToA(dtStruct->hour,(unsigned long)&(((char*)pString)[12]),BRDK_STR_CONVERT_DECIMAL);
	}
	else brdkStrUdintToA(dtStruct->hour,(unsigned long)&(((char*)pString)[11]),BRDK_STR_CONVERT_DECIMAL);
	((char*)pString)[13] = BRDK_STR_ASCII_COLON;
	if(dtStruct->minute < 10) {
		((char*)pString)[14] = BRDK_STR_ASCII_0;
		brdkStrUdintToA(dtStruct->minute,(unsigned long)&(((char*)pString)[15]),BRDK_STR_CONVERT_DECIMAL);
	}
	else brdkStrUdintToA(dtStruct->minute,(unsigned long)&(((char*)pString)[14]),BRDK_STR_CONVERT_DECIMAL);
	((char*)pString)[16] = BRDK_STR_ASCII_COLON;
	if(dtStruct->second < 10) {
		((char*)pString)[17] = BRDK_STR_ASCII_0;
		brdkStrUdintToA(dtStruct->second,(unsigned long)&(((char*)pString)[18]),BRDK_STR_CONVERT_DECIMAL);
	}
	else brdkStrUdintToA(dtStruct->second,(unsigned long)&(((char*)pString)[17]),BRDK_STR_CONVERT_DECIMAL);
	((char*)pString)[19] = BRDK_STR_ASCII_DOT;
	if(dtStruct->millisec < 10) {
		((char*)pString)[20] = BRDK_STR_ASCII_0;
		((char*)pString)[21] = BRDK_STR_ASCII_0;
		brdkStrUdintToA(dtStruct->millisec,(unsigned long)&(((char*)pString)[22]),BRDK_STR_CONVERT_DECIMAL);
	}
	else if(dtStruct->millisec < 100) {
		((char*)pString)[20] = BRDK_STR_ASCII_0;
		brdkStrUdintToA(dtStruct->millisec,(unsigned long)&(((char*)pString)[21]),BRDK_STR_CONVERT_DECIMAL);
	}
	else brdkStrUdintToA(dtStruct->millisec,(unsigned long)&(((char*)pString)[20]),BRDK_STR_CONVERT_DECIMAL);
	((char*)pString)[23] = BRDK_STR_ASCII_NULL;
	return 23;
}
```

#### brdkStrEncode.c
```c
#include <brdkSTR_func.h>

signed long brdkStrEncode(unsigned long pDestination, unsigned long pSource, unsigned char format) {
	unsigned long i=0;
	switch(format) {
		case BRDK_STR_UTF_8:

			do ((unsigned char*)pDestination)[i] = ((unsigned char*)pSource)[i] <= 127 ? ((unsigned char*)pSource)[i] : ((unsigned char*)pSource)[i] + 35;
			while(((char*)pSource)[i++] != BRDK_STR_ASCII_NULL);
			return pDestination+i;
			break;

		default:
			return -1;
			break;
	}
}
```

#### brdkStrFill.c
```c
#include <brdkSTR_func.h>

signed long brdkStrFill(unsigned long pString, signed long amount, unsigned long pChar, signed long position) {
	signed long i,j, len = brdkStrLen(pString), tmpPos;
	char ch;
	i = len+amount;
	j = len;
	ch = pChar != 0 && *(char*)pChar != BRDK_STR_ASCII_NULL ? *(char*)pChar : BRDK_STR_ASCII_SPACE;	/* white space is default */
	tmpPos = position >= 0 ? position : len + 1 + position;
	if(tmpPos > -1) {
		while(j>=tmpPos) ((char*)pString)[i--] = ((char*)pString)[j--];
		while(i>=tmpPos) ((char*)pString)[i--] = ch;
		return len+amount;
	}
	else return -1;
}
```

#### brdkStrFillUp.c
```c
#include <brdkSTR_func.h>

signed long brdkStrFillUp(unsigned long pString, signed long maxLength, unsigned long pChar, signed long position) {
	signed long amount = maxLength-brdkStrLen(pString);
	if(amount > 0) {
		if(brdkStrFill(pString, amount, pChar, position) != -1) return amount;
		else return -1;
	}
	return 0;
}
```

#### brdkStrIndexOf.c
```c
#include <brdkSTR_func.h>

signed long brdkStrIndexOf(unsigned long pString, unsigned long pChar, signed long direction) {
	signed long i;
	if(direction > -1) {
		i = 0;
		while(((char*)pString)[i]) {
			if(((char*)pString)[i] == ((char*)pChar)[0]) break;
			else i++;
		}
		if(((char*)pString)[i] != BRDK_STR_ASCII_NULL) return i;
		else return -1;
	}
	else {
		i = brdkStrLen(pString)-1;
		while(((char*)pString)[i] && i > -1) if(((char*)pString)[i--] == ((char*)pChar)[0]) break;
		if(((char*)pString)[i] != BRDK_STR_ASCII_NULL) return ++i;
		else return -1;
	}
}
```

#### brdkStrInsertAtPos.c
```c
#include <brdkSTR_func.h>

signed long brdkStrInsertAtPos(unsigned long pString, unsigned long pInsert, signed long position) {
	signed long i,j, len = brdkStrLen(pString), lenIns = brdkStrLen(pInsert), tmpPos;
	if(lenIns > 0) {
		if(len==0 && (position==0 || position==-1)){
			i=0;
			while(((char*)pInsert)[i]) {
				((char*)pString)[i] = ((char*)pInsert)[i];
				i++;
			}
			((char*)pString)[i] = BRDK_STR_ASCII_NULL;
			len = i;
		}
		else if(position <= len) {
			i = len+lenIns;
			j = len;
			tmpPos = position >= 0 ? position : len + 1 + position;
			if(tmpPos > -1) {
				while(j>=tmpPos) ((char*)pString)[i--] = ((char*)pString)[j--];
				j=lenIns-1;
				while(i>=tmpPos) ((char*)pString)[i--] = ((char*)pInsert)[j--];
				len+=lenIns;
			}
			else len = -1;
		}
	}
	return len;
}
```

#### brdkStrIsAlphabet.c
```c
#include <brdkSTR_func.h>

unsigned char brdkStrIsAlphabet(unsigned long pString) {
	unsigned long len = 0;
	while(((char*)pString)[len]) {
		if (((char*)pString)[len] > BRDK_STR_ASCII_Z) {
			if(((char*)pString)[len] < BRDK_STR_ASCII_a || BRDK_STR_ASCII_z < ((char*)pString)[len]) return 0;
		}
		else if(((char*)pString)[len] < BRDK_STR_ASCII_A) return 0;
		len++;
	}
	return 1;
}
```

#### brdkStrIsDigit.c
```c
#include <brdkSTR_func.h>

unsigned char brdkStrIsDigit(unsigned long pString) {
	unsigned long len = 0;
	while(((char*)pString)[len]) {
		if (((char*)pString)[len] < BRDK_STR_ASCII_0 || BRDK_STR_ASCII_9 < ((char*)pString)[len]) return 0;
		len++;
	}
	return 1;
}
```

#### brdkStrIsEmpty.c
```c
#include <brdkSTR_func.h>

unsigned char brdkStrIsEmpty(unsigned long pString) {
	return ((char*)pString)[0] == BRDK_STR_ASCII_NULL;
}
```

#### brdkStrJoin.c
```c
#include <brdkSTR_func.h>

signed long brdkStrJoin(unsigned long pString, unsigned long pArray, unsigned long pDelimiter, unsigned long sizeOfArray, unsigned long sizeOfArrayString, unsigned long sizeOfString) {
	unsigned long sIdx = 0, pArr = pArray, aIdx = 0;
	if(pArray != 0 && pString != 0 && sizeOfArray != 0 && sizeOfArrayString != 0) {		/* check all pointers are set */
		if(pDelimiter == 0) pDelimiter = (unsigned long)" ";							/* use white space is delimiter pointer is 0 */
		while(((char*)pArr)[0] != 0) {													/* continue until we find the first empty array string */
			if(((char*)pArr)[aIdx] != 0) {
				((char*)pString)[sIdx++] = ((char*)pArr)[aIdx++];						/* copy string data */
				if(sIdx >= sizeOfString) return -2;										/* destination string too small */
			}
			else {
				pArr += sizeOfArrayString;												/* jump to the next array element */
				aIdx = 0;
				((char*)pString)[sIdx++] = ((char*)pDelimiter)[0];						/* insert delimiter */
				if(sIdx >= sizeOfString) return -2;										/* destination string too small */
				if(pArr > (pArray + sizeOfArray)) {										/* we hit the end of the array */
					break;
				}
			}
		}
		if(sIdx == 0) return 0;															/* nothing copied */
		sIdx--;
		((char*)pString)[sIdx] = 0;														/* end the string. -e because we inserted a delimiter at the end */
		return sIdx;
	}
	else return -1;
	return -4;
}
```

#### brdkStrLen.c
```c
#include <brdkSTR_func.h>

signed long brdkStrLen(unsigned long pString) {
	unsigned long len = 0;
	while(((char*)pString)[len]) len++;	/* makes a little strlen */
	return len;
}
```

#### brdkStrMemClear.c
```c
#include <brdkSTR_func.h>

unsigned long brdkStrMemClear(unsigned long pDestination, unsigned long amount) {
	return brdkStrMemSet(pDestination,0,amount);
}
```

#### brdkStrMemCmp.c
```c
#include <brdkSTR_func.h>

signed long brdkStrMemCmp(unsigned long pString1, unsigned long pString2, unsigned long amount) {
	unsigned long i=0;
	for(i=0; i< amount; i++) if(((char*)pString1)[i] != ((char*)pString2)[i]) break;
	return ((char*)pString1)[i]-((char*)pString2)[i];
}
```

#### brdkStrMemCpy.c
```c
#include <brdkSTR_func.h>

unsigned long brdkStrMemCpy(unsigned long pDestination, unsigned long pSource, unsigned long amount) {
	unsigned long i=0;
	for(i=0; i< amount; i++) ((char*)pDestination)[i] = ((char*)pSource)[i];
	return pDestination+amount;
}
```

#### brdkStrMemMove.c
```c
#include <brdkSTR_func.h>

unsigned long brdkStrMemMove(unsigned long pDestination, unsigned long pSource, unsigned long amount) {
	unsigned long i=0;
	char buffer[amount];	/* if the destination and source is the same string we need a buffer */
	for(i=0; i< amount; i++) buffer[i] = ((char*)pSource)[i];
	for(i=0; i< amount; i++) ((char*)pDestination)[i] = buffer[i];
	return pDestination+amount;
}
```

#### brdkStrMemSet.c
```c
#include <brdkSTR_func.h>

unsigned long brdkStrMemSet(unsigned long pDestination, unsigned char value, unsigned long amount) {
	unsigned long i=0;
	for(i=0; i< amount; i++) ((char*)pDestination)[i] = value;
	return pDestination+amount;
}
```

#### brdkStrMove.c
```c
#include <brdkSTR_func.h>

unsigned long brdkStrMove(unsigned long pDestination, unsigned long pSource) {
	return brdkStrMemMove(pDestination,pSource,brdkStrLen(pSource));
}
```

#### brdkStrNAToDint.c
```c
#include <brdkSTR_func.h>

signed long brdkStrNAToDint(unsigned long pString, unsigned long amount, unsigned char base) {
	/* check if string starts with a hypen */
	if(amount == 0) return 0;
	if(((char*)pString)[0] == BRDK_STR_ASCII_HYPHEN) return -brdkStrNAToUdint(pString+1,amount-1, BRDK_STR_CONVERT_DECIMAL);
	else return brdkStrNAToUdint(pString, amount, base);
}
```

#### brdkStrNAToUdint.c
```c
#include <brdkSTR_func.h>

unsigned long brdkStrNAToUdint(unsigned long pString, unsigned long amount, unsigned char base) {
	unsigned long value = 0,i;
	if(amount > 0) {
		for(i=0; i < amount; i++) {
			switch(base) {

				case 0: case 10:
					if(((char*)pString)[i] >= BRDK_STR_ASCII_0 && ((char*)pString)[i] <= BRDK_STR_ASCII_9) value = (value * 10) + (((char*)pString)[i]-BRDK_STR_ASCII_0);			/* 0x30 = 0, 0x39 = 9 */
					else {
						value = 0;
						i = amount;
					}
					break;

				case 2:
					if(((char*)pString)[i] >= BRDK_STR_ASCII_0 && ((char*)pString)[i] <= BRDK_STR_ASCII_1) value += (((char*)pString)[i]-BRDK_STR_ASCII_0)*(1<<(amount-1-i));			/* 0x30 = 0, 0x31 = 1 */
					else {
						value = 0;
						i = amount;
					}
					break;

				case 16:
					if(((char*)pString)[i] >= BRDK_STR_ASCII_0 && ((char*)pString)[i] <= BRDK_STR_ASCII_9) 	value += (((char*)pString)[i]-BRDK_STR_ASCII_0)*(1<<(4*(amount-1-i)));		/* 0x30 = 0, 0x39 = 9 */
					else if(((char*)pString)[i] >= BRDK_STR_ASCII_A && ((char*)pString)[i] <= BRDK_STR_ASCII_F) value += (((char*)pString)[i]-BRDK_STR_ASCII_7)*(1<<(4*(amount-1-i)));	/* 0x41 = A, 0x46 = F */
					else if(((char*)pString)[i] >= BRDK_STR_ASCII_a && ((char*)pString)[i] <= BRDK_STR_ASCII_f)value += (((char*)pString)[i]-BRDK_STR_ASCII_W)*(1<<(4*(amount-1-i)));	/* 0x61 = a, 0x66 = f */
					else {
						value = 0;
						i = amount;
					}
					break;

				default:
					value = 0;
					i = amount;
					break;

			}
		}
	}
	return value;
}
```

#### brdkStrNCpy.c
```c
#include <brdkSTR_func.h>

unsigned long brdkStrNCpy(unsigned long pDestination, unsigned long pSource, unsigned long amount) {
	unsigned long i=0;
	for(i=0; i< amount; i++) {
		if(((char*)pSource)[i]) ((char*)pDestination)[i] = ((char*)pSource)[i];
		else ((char*)pDestination)[i] = BRDK_STR_ASCII_NULL;
	}
	return pDestination+amount;
}
```

#### brdkStrNIsAlphabet.c
```c
#include <brdkSTR_func.h>

unsigned char brdkStrNIsAlphabet(unsigned long pString, unsigned long amount) {
	unsigned long i = 0;
	for(; i < amount; i++) {
		if(((char*)pString)[i] > BRDK_STR_ASCII_Z) {
			if(((char*)pString)[i] < BRDK_STR_ASCII_a || BRDK_STR_ASCII_z < ((char*)pString)[i]) return 0;
		}
		else if(((char*)pString)[i] < BRDK_STR_ASCII_A) return 0;
	}
	return 1;
}
```

#### brdkStrNIsDigit.c
```c
#include <brdkSTR_func.h>

unsigned char brdkStrNIsDigit(unsigned long pString, unsigned long amount) {
	unsigned long i = 0;
	for(;i < amount; i++) if (((char*)pString)[i] < BRDK_STR_ASCII_0 || BRDK_STR_ASCII_9 < ((char*)pString)[i]) return 0;
	return 1;
}
```

#### brdkStrRemove.c
```c
#include <brdkSTR_func.h>

unsigned long brdkStrRemove(unsigned long pString, signed long start, signed long length) {
	signed long end, len=0;
	if(start < 0) {
		len = brdkStrLen(pString);
		if(length<1) {
			len = start;
			start = length*(-1);
			length = brdkStrLen(pString)-start+len+1;
		}
		else start = len+start-length+1;
	}
	else if(length<1) length = brdkStrLen(pString)-start+length;
	end = start+length;
	while(((char*)pString)[end]) ((char*)pString)[start++] = ((char*)pString)[end++];
	((char*)pString)[start] = BRDK_STR_ASCII_NULL;
	return pString+start+1;
}
```

#### brdkStrRepeat.c
```c
#include <brdkSTR_func.h>

signed long brdkStrRepeat(unsigned long pString, signed long times) {
	signed long i,j,t,len = brdkStrLen(pString);
	j=len;
	for(t=0; t < times; t++) {
		for(i=0; i< len; i++) ((char*)pString)[j+i] = ((char*)pString)[i];
		j += len;
	}
	((char*)pString)[j] = BRDK_STR_ASCII_NULL;
	return j;
}
```

#### brdkStrReplace.c
```c
#include <brdkSTR_func.h>

signed long brdkStrReplace(unsigned long pString, unsigned long pFind, unsigned long pReplace) {
	signed long i=0, cnt=0, lenF = brdkStrLen(pFind), lenR = brdkStrLen(pReplace);
	i = brdkStrSearch(pString,pFind);
	while(i > -1) {
		brdkStrRemove(pString,i,lenF);
		brdkStrInsertAtPos(pString,pReplace,i);
		pString += i + lenR;
		i = brdkStrSearch(pString,pFind);
		cnt++;
	}
	return cnt;
}
```

#### brdkStrReverse.c
```c
#include <brdkSTR_func.h>

signed long brdkStrReverse(unsigned long pString, signed long startPosition, signed long endPosition) {
	signed long start = -1, end = -1, len = brdkStrLen(pString), cnt = 0;
    unsigned char tmp;
	/* make sure start position is valid */
	if(startPosition > -1 && startPosition < len) start = startPosition;
	else return -1;
	/* make sure end position is valid */
	if(endPosition > -1 && endPosition < len && endPosition > startPosition) end = endPosition;
	else if(endPosition < 0) end = len + endPosition;
	else return -1;
	while (start < end) {
        tmp = ((char*)pString)[start];
        ((char*)pString)[start++] = ((char*)pString)[end];
        ((char*)pString)[end--] = tmp;
		cnt++;
    }
	return cnt;
}
```

#### brdkStrReverseWords.c
```c
#include <brdkSTR_func.h>

signed long brdkStrReverseWords(unsigned long pString) {
	signed long i=0,wordPos=-1, cnt=0;
	while(((char*)pString)[i]) {
		if(wordPos<0 && (((char*)pString)[i] != BRDK_STR_ASCII_SPACE)) wordPos = i;
		if(wordPos>-1 && (((char*)pString)[i+1] == BRDK_STR_ASCII_SPACE || ((char*)pString)[i+1] == 0)) {
			brdkStrReverse(pString,wordPos,i);
            wordPos = -1;
			cnt++;
        }
		i++;
	}
	brdkStrReverse(pString,0,i-1);
	return cnt;
}
```

#### brdkStrSearch.c
```c
#include <brdkSTR_func.h>

signed long brdkStrSearch(unsigned long pString, unsigned long pSearchString) {
	signed long lenString = brdkStrLen(pString), lenSearch = brdkStrLen(pSearchString);
	return search(pString, lenString, pSearchString, lenSearch);
}
```

#### brdkStrSlice.c
```c
#include <brdkSTR_func.h>

signed long brdkStrSlice(unsigned long pString, signed long start, signed long end) {
	signed long i,j, len = -1;
	if(start > -1) {
		if(start > 0) {
			len = brdkStrLen(pString);
			j=0;
			while(j<start) {
				for(i=0;i < len;i++) ((char*)pString)[i] = ((char*)pString)[i+1];	/* moves all characters one place left */
				len--;
				j++;
			}
		}
		if(end > 0) {
			end -= start;
			((char*)pString)[end] = BRDK_STR_ASCII_NULL;
			len = end;
		}
		else if(end < 0) {
			len = brdkStrLen(pString);
			if((end*(-1))<=len) {
				len += end;
				((char*)pString)[len+1+end] = BRDK_STR_ASCII_NULL;
			}
		}
		return len;
	}
	else return -1;
}
```

#### brdkStrSplit.c
```c
#include <brdkSTR_func.h>

signed long brdkStrSplit(unsigned long pArray, unsigned long pString, unsigned long pDelimiter, unsigned long sizeOfArray, unsigned long sizeOfArrayString, unsigned char greedy) {
	signed long size = 0;
	if(pArray != 0 && pString != 0 && sizeOfArray != 0 && sizeOfArrayString != 0) {		/* check all pointers are set */
		if(pDelimiter == 0) pDelimiter = (unsigned long)" ";							/* use white space is delimiter pointer is 0 */
		unsigned long i = 0, pArr = pArray, aIdx = 0;
		while(((char*)pString)[i] != 0) {												/* run while we dopn't hit a 0 */
			if(((char*)pString)[i] != ((char*)pDelimiter)[0]) {							/* check for delimiter */
				((char*)pArr)[aIdx++] = ((char*)pString)[i++];
				if(aIdx >= sizeOfArrayString) return -2;								/* array string too small */
			}
			else {
				if(!greedy) ((char*)pArr)[aIdx++] = ((char*)pString)[i];				/* check is delimiter should be removed */
				i++;
				if(aIdx >= sizeOfArrayString) return -2;								/* array string too small */
				((char*)pArr)[aIdx] = BRDK_STR_ASCII_NULL;
				pArr += sizeOfArrayString;												/* jump to the next array element */
				aIdx = 0;
				size++;
				if(pArr > (pArray + sizeOfArray)) return -3;							/* array too small */
			}
		}
		((char*)pArr)[aIdx] = BRDK_STR_ASCII_NULL;
		pArr += sizeOfArrayString;														/* jump to the next array element */
		size++;
		while(pArr < (pArray + sizeOfArray)) {											/* set the rest of the array elements to '' */
			((char*)pArr)[0] = BRDK_STR_ASCII_NULL;
			pArr += sizeOfArrayString;
		}
		return size;
	}
	else return -1;
	return -4;
}
```

#### brdkStrSubDintSearch.c
```c
#include <brdkSTR_func.h>

signed long brdkStrSubDintSearch(unsigned long pSource, unsigned long pStart, unsigned long pEnd, signed long startOffset, unsigned char base) {
	signed long posEnd, lenSource = brdkStrLen(pSource), lenStart = brdkStrLen(pStart), lenEnd, posGreedyStartOffset;
	signed long posStart = search(pSource, lenSource, pStart, lenStart);
	if(posStart > -1) {
		lenEnd = brdkStrLen(pEnd);
		posGreedyStartOffset = posStart + lenStart + startOffset;
		posEnd = search((unsigned long)&((char*)pSource)[posGreedyStartOffset], lenSource-posGreedyStartOffset, pEnd, lenEnd);
		if(posEnd > -1) {
			/* check if string starts with a hyphen */
			if(((char*)pSource)[posGreedyStartOffset] == BRDK_STR_ASCII_HYPHEN) return -brdkStrNAToUdint((unsigned long)&((char*)pSource)[posGreedyStartOffset+1],posEnd,base);
			else return brdkStrNAToUdint((unsigned long)&((char*)pSource)[posGreedyStartOffset],posEnd,base);
		}
	}
	return -1;
}
```

#### brdkStrSubStr.c
```c
#include <brdkSTR_func.h>

signed long brdkStrSubStr(unsigned long pDestination, unsigned long pSource, signed long start, signed long length) {
	signed long i=0,len=0;
	char buffer[length];	/* if the destination and source is the same string we need a buffer */
	if(start < 0) {
		len = brdkStrLen(pSource);
		if(length<1) {
			len = start;
			start = length*(-1);
			length = brdkStrLen(pSource)-start+len+1;
		}
		else start = len+start-length+1;
	}
	else if(length<1) length = brdkStrLen(pSource)-start+length;
	for(i=0; i< length; i++) buffer[i] = ((char*)pSource)[start+i];
	for(i=0; i< length; i++) ((char*)pDestination)[i] = buffer[i];
	((char*)pDestination)[i] = BRDK_STR_ASCII_NULL;
	return length;
}
```

#### brdkStrSubStrSearch.c
```c
#include <brdkSTR_func.h>

unsigned char brdkStrSubStrSearch(unsigned long pDestination, unsigned long pSource, unsigned long pStart, unsigned long pEnd, signed long startOffset, unsigned char greedy) {
	signed long posEnd, lenSource = brdkStrLen(pSource), lenStart = brdkStrLen(pStart), lenEnd, posGreedyStartOffset;
	signed long posStart = search(pSource, lenSource, pStart, lenStart);
	if(posStart > -1) {
		lenEnd = brdkStrLen(pEnd);
		posGreedyStartOffset = posStart + lenStart + startOffset;
		posEnd = search((unsigned long)&((char*)pSource)[posGreedyStartOffset], lenSource-posGreedyStartOffset, pEnd, lenEnd);
		if(posEnd > -1) {
			if(!greedy) {
				posGreedyStartOffset = posStart;
				posEnd += lenStart + startOffset + 1;
			}
			brdkStrMemCpy(pDestination, (unsigned long)&((char*)pSource)[posGreedyStartOffset],posEnd);
			((char*)pDestination)[posEnd] = BRDK_STR_ASCII_NULL;
			return 1;
		}
	}
	return 0;
}
```

#### brdkStrToDec.c
```c
#include <brdkSTR_func.h>

signed long brdkStrToDec(unsigned long pString) {
	signed long i=0,j=0;
	while(((char*)pString)[i]) {
		if(((char*)pString)[i+1] != BRDK_STR_ASCII_NULL) {
			char tmp[3];
			tmp[0] = ((char*)pString)[i++];
			tmp[1] = ((char*)pString)[i++];
			tmp[2] = 0;
			((char*)pString)[j++] = brdkStrAToUdint((unsigned long)&tmp, BRDK_STR_CONVERT_HEX);
		}
		else {
			i = -1;
			break;
		}
		((char*)pString)[j] = BRDK_STR_ASCII_NULL;
	}
	return i;
}
```

#### brdkStrToHex.c
```c
#include <brdkSTR_func.h>

signed long brdkStrToHex(unsigned long pString) {
	signed long i=0;
	unsigned long rem;
	unsigned char tmp;
	while(((char*)pString)[i]) {
		unsigned char value = (unsigned char)((char*)pString)[i];
		if(value < 0x10) {															/* a character with value below 9 we want representated with a 0 in front */
			brdkStrFill(pString,1,(unsigned long)&"0",i++);
			rem = value % 16;
		    ((char*)pString)[i++] = (rem > 9)? (rem-10) + BRDK_STR_ASCII_A : rem + BRDK_STR_ASCII_0;
		}
		else {
			while(value > 0) {
				rem = value % 16;
		       	((char*)pString)[i++] = (rem > 9)? (rem-10) + BRDK_STR_ASCII_A : rem + BRDK_STR_ASCII_0;
		       	value = value/16;
				if(value > 0) brdkStrFill(pString,1,(unsigned long)&" ",i);
				else {
					/* swap places */
					tmp = ((char*)pString)[i-1];
					((char*)pString)[i-1] = ((char*)pString)[i-2];
					((char*)pString)[i-2] = tmp;
				}
			}
		}
	}
	((char*)pString)[i] = BRDK_STR_ASCII_NULL;
	return i;
}
```

#### brdkStrToLowerCase.c
```c
#include <brdkSTR_func.h>

signed long brdkStrToLowerCase(unsigned long pString) {
	unsigned long i=0, cnt=0;
	while(((char*)pString)[i]) {
		if((((char*)pString)[i] >= BRDK_STR_ASCII_A) && (((char*)pString)[i] <= BRDK_STR_ASCII_Z)) {	/* between A..Z */
			((char*)pString)[i] += BRDK_STR_ASCII_SPACE;
			cnt++;
		}
		i++;
	}
	return cnt;
}
```

#### brdkStrToUpperCase.c
```c
#include <brdkSTR_func.h>

signed long brdkStrToUpperCase(unsigned long pString) {
	unsigned long i=0,cnt=0;
	while(((char*)pString)[i]) {
		if((((char*)pString)[i] >= BRDK_STR_ASCII_a) && (((char*)pString)[i] <= BRDK_STR_ASCII_z)) {	/* between a..z */
			((char*)pString)[i] -= BRDK_STR_ASCII_SPACE;
			cnt++;
		}
		i++;
	}
	return cnt;
}
```

#### brdkStrToUpperCaseWords.c
```c
#include <brdkSTR_func.h>

signed long brdkStrToUpperCaseWords(unsigned long pString) {
	unsigned long i=0,cnt=0;
	if(((char*)pString)[i]) {
		if(((char*)pString)[i] >= BRDK_STR_ASCII_a && ((char*)pString)[i] <= BRDK_STR_ASCII_z) {	/* check the first character */
	 		((char*)pString)[i] -= BRDK_STR_ASCII_SPACE;
			cnt++;
		}
	}
	i++;
	while(((char*)pString)[i]) {
		if((((char*)pString)[i] >= BRDK_STR_ASCII_a) && (((char*)pString)[i] <= BRDK_STR_ASCII_z) && ((char*)pString)[i-1] == BRDK_STR_ASCII_SPACE){	/* between a..z and a space before */
			((char*)pString)[i] -= BRDK_STR_ASCII_SPACE;
			cnt++;
		}
		i++;
	}
	return cnt;
}
```

#### brdkStrTrim.c
```c
#include <brdkSTR_func.h>

signed long brdkStrTrim(unsigned long pString, signed long direction) {
	signed long i,j=0,len;
	if(direction == BRDK_STR_BOTH_TRIM || direction == BRDK_STR_LEFT_TRIM) {
		len = brdkStrLen(pString);
		while(((char*)pString)[0] == BRDK_STR_ASCII_SPACE) {
			for(i=0;i < len;i++) ((char*)pString)[i] = ((char*)pString)[i+1];	/* moves all characters one place left */
			len--;
			j++;
		}
	}
	if(direction == BRDK_STR_BOTH_TRIM || direction == BRDK_STR_RIGHT_TRIM) {
		len = brdkStrLen(pString)-1;
		while(((char*)pString)[len] == BRDK_STR_ASCII_SPACE && len > -1) {
			((char*)pString)[len--] = BRDK_STR_ASCII_NULL;
			j++;
		}
	}
	return j;
}
```

#### brdkStrUdintToA.c
```c
#include <brdkSTR_func.h>

signed long brdkStrUdintToA(unsigned long value, unsigned long pString, unsigned char base) {
	int i=0;
	((char*)pString)[0] = 0;
	base = !base ? 10 : base;	/* make sure base is not 0 */
	if (value != 0) {
		while (value > 0) {
			unsigned long rem = value % base;
	       	((char*)pString)[i++] = (rem > 9)? (rem-10) + BRDK_STR_ASCII_A : rem + BRDK_STR_ASCII_0;
	       	value = value/base;
		}
		((char*)pString)[i] = BRDK_STR_ASCII_NULL;
	}
	else {
		((char*)pString)[i++] = BRDK_STR_ASCII_0;
		((char*)pString)[i] = BRDK_STR_ASCII_NULL;
	}
	brdkStrReverse(pString,0,-1);
	return i;
}
```

#### brdkStrWord.c
```c
#include <brdkSTR_func.h>

signed long brdkStrWord(unsigned long pDestination, unsigned long pSource, unsigned long pDelimiter, signed long number, unsigned long sizeOfString) {
	unsigned long sIdx = 0, dIdx = 0;
	signed long cnt = 1;
	if(pDestination != 0 && pSource != 0 && number != 0) {
		if(pDelimiter == 0) pDelimiter = (unsigned long)" ";			/* use white space is delimiter pointer is 0 */
		while(((char*)pSource)[sIdx] != 0) {
			if(((char*)pSource)[sIdx] != ((char*)pDelimiter)[0]) {
				((char*)pDestination)[dIdx++] = ((char*)pSource)[sIdx];
			}
			else {
				if(number > 0) {
					if(cnt == number) break;
					else {
						dIdx = 0;
						cnt++;
					}
				}
				else {
					cnt = number;
					dIdx = 0;
				}
			}
			sIdx++;
			if(dIdx > sizeOfString) return -2;								/* destination string too small */
		}
		if(number > cnt) return -3;
		((char*)pDestination)[dIdx] = BRDK_STR_ASCII_NULL;
		return dIdx;
	}
	else return -1;
	return -4;
}
```

#### brdkSTR_func.h
```c
#ifndef BRDK_STR_FUNCS
#define BRDK_STR_FUNCS 1

#include <brdkSTR.h>
#include <bur/plctypes.h>

#ifdef __cplusplus
	extern "C"
	{
#endif

signed long search(signed long pString, signed long lenString, signed long pSearchString, signed long lenSearch);
unsigned char dayOfWeek(unsigned char d,unsigned char m, unsigned short y);

#ifdef __cplusplus
	};
#endif

#endif
```

#### brdkSTR_func.c
```c
#include <brdkSTR_func.h>

/* search for a string in a string */
signed long search(signed long pString, signed long lenString, signed long pSearchString, signed long lenSearch) {
	signed long pos=-1, i=0,j=0;
	if(lenString>lenSearch) {
		for(i=0; i <= lenString-lenSearch; i++) {
			j=0;
			if(((char*)pString)[i] == ((char*)pSearchString)[j]) {
				while(((char*)pString)[i+j] == ((char*)pSearchString)[j]) {
					j++;
					if(j==lenSearch) {
						pos = i;
						i=lenString-lenSearch+1;
						break;
					}
				}
			}
		}
	}
	return pos;
}

unsigned char dayOfWeek(unsigned char d,unsigned char m, unsigned short y){
	unsigned char t[] = { 0, 3, 2, 5, 0, 3, 5, 1, 4, 6, 2, 4 };
	if (m < 3) y -= 1;
	return((y + y / 4 - y / 100 + y / 400 + t[m - 1] + d) % 7);
}
```

- CHANGELOG - brdkSTR change log (not shown)

- LICENSE - brdkSTR license (not shown)

### Library Logical/Libraries/PackMLCore (ANSIC, version 1.1.1)

#### PackMLModule.hpp
```cpp
#ifndef __PACKMLMODULE_HPP__
#define __PACKMLMODULE_HPP__

#include "PackMLModuleEnums.hpp"
#include <vector>
#include <string>
#include <string.h>
//#include <cmath>
#include "AtomicSemaphore.hpp"
#include "PackMLModuleSharedInfo.hpp"

		// PackMLModule main class
class PackMLModule {

	public:
	PackMLModule(const char* pModuleName);
	~PackMLModule();

	// *** onCreated() ***
	// root module
	void initModule();
	// child module
	bool initModule(PackMLModule* pParent);

	// *** onBeforeShutdown() ***
	bool exitModule();

	// *** run() ***
	void runPackMLModule();

	// **********************************************************
	// ************* Real time parameter update *****************
	// **********************************************************
	void setActivationCondition(short int newParameter){
		activationCondition_ = newParameter;
	}

	void setOverrideAbort(bool newParameter)
	{
		overrideAbort_ = newParameter && (hierarchyLevel_ > 0);
	}
	void setOverrideStop(bool newParameter)
	{
		overrideStop_ = newParameter && (hierarchyLevel_ > 0);
	}
	void setOverrideClear(bool newParameter)
	{
		overrideClear_ = newParameter && (hierarchyLevel_ > 0);
	}
	void setOverrideReset(bool newParameter)
	{
		overrideReset_ = newParameter && (hierarchyLevel_ > 0);
	}
	void setOverrideStart(bool newParameter)
	{
		overrideStart_ = newParameter && (hierarchyLevel_ > 0);
	}
	void setOverrideSuspend(bool newParameter)
	{
		overrideSuspend_ = newParameter && (hierarchyLevel_ > 0);
	}
	void setOverrideUnsuspend(bool newParameter)
	{
		overrideUnsuspend_ = newParameter && (hierarchyLevel_ > 0);
	}
	void setOverrideHold(bool newParameter)
	{
		overrideHold_ = newParameter && (hierarchyLevel_ > 0);
	}
	void setOverrideUnhold(bool newParameter)
	{
		overrideUnhold_ = newParameter && (hierarchyLevel_ > 0);
	}
	void setOverrideComplete(bool newParameter)
	{
		overrideComplete_ = newParameter && (hierarchyLevel_ > 0);
	}

	void setReactToAbort(bool newParameter)
	{
		reactToAbort_ = newParameter && (hierarchyLevel_ > 0);
	}
	void setReactToStop(bool newParameter)
	{
		reactToStop_ = newParameter && (hierarchyLevel_ > 0);
	}
	void setReactToClear(bool newParameter)
	{
		reactToClear_ = newParameter && (hierarchyLevel_ > 0);
	}
	void setReactToReset(bool newParameter)
	{
		reactToReset_ = newParameter && (hierarchyLevel_ > 0);
	}
	void setReactToStart(bool newParameter)
	{
		reactToStart_ = newParameter && (hierarchyLevel_ > 0);
	}
	void setReactToSuspend(bool newParameter)
	{
		reactToSuspend_ = newParameter && (hierarchyLevel_ > 0);
	}
	void setReactToUnsuspend(bool newParameter)
	{
		reactToUnsuspend_ = newParameter && (hierarchyLevel_ > 0);
	}
	void setReactToHold(bool newParameter)
	{
		reactToHold_ = newParameter && (hierarchyLevel_ > 0);
	}
	void setReactToUnhold(bool newParameter)
	{
		reactToUnhold_ = newParameter && (hierarchyLevel_ > 0);
	}
	void setReactToComplete(bool newParameter)
	{
		reactToComplete_ = newParameter && (hierarchyLevel_ > 0);
	}

	void setEscalateAbort(bool newParameter)
	{
		escalateAbort_ = newParameter && (hierarchyLevel_ > 0);
	}
	void setEscalateStop(bool newParameter)
	{
		escalateStop_ = newParameter && (hierarchyLevel_ > 0);
	}
	void setEscalateClear(bool newParameter)
	{
		escalateClear_ = newParameter && (hierarchyLevel_ > 0);
	}
	void setEscalateReset(bool newParameter)
	{
		escalateReset_ = newParameter && (hierarchyLevel_ > 0);
	}
	void setEscalateStart(bool newParameter)
	{
		escalateStart_ = newParameter && (hierarchyLevel_ > 0);
	}
	void setEscalateSuspend(bool newParameter)
	{
		escalateSuspend_ = newParameter && (hierarchyLevel_ > 0);
	}
	void setEscalateUnsuspend(bool newParameter)
	{
		escalateUnsuspend_ = newParameter && (hierarchyLevel_ > 0);
	}
	void setEscalateHold(bool newParameter)
	{
		escalateHold_ = newParameter && (hierarchyLevel_ > 0);
	}
	void setEscalateUnhold(bool newParameter)
	{
		escalateUnhold_ = newParameter && (hierarchyLevel_ > 0);
	}
	void setEscalateComplete(bool newParameter)
	{
		escalateComplete_ = newParameter && (hierarchyLevel_ > 0);
	}

	bool evaluateCmdAbort(bool& newCmd);
	bool evaluateCmdStop(bool& newCmd);
	bool evaluateCmdClear(bool& newCmd);
	bool evaluateCmdReset(bool& newCmd);
	bool evaluateCmdStart(bool& newCmd);
	bool evaluateCmdSuspend(bool& newCmd);
	bool evaluateCmdUnsuspend(bool& newCmd);
	bool evaluateCmdHold(bool& newCmd);
	bool evaluateCmdUnhold(bool& newCmd);
	bool evaluateCmdComplete(bool& newCmd);
	bool evaluateCmdStateComplete(bool& newCmd);

	bool setCmdAbort();
	bool setCmdStop();
	bool setCmdClear();
	bool setCmdReset();
	bool setCmdStart();
	bool setCmdSuspend();
	bool setCmdUnsuspend();
	bool setCmdHold();
	bool setCmdUnhold();
	bool setCmdComplete();
	bool setCmdStateComplete();

	bool getCmdAbort(){
		return abort_;
	}
	bool getCmdStop(){
		return stop_;
	}
	bool getCmdClear(){
		return clear_;
	}
	bool getCmdReset(){
		return reset_;
	}
	bool getCmdStart(){
		return start_;
	}
	bool getCmdSuspend(){
		return suspend_;
	}
	bool getCmdUnsuspend(){
		return unsuspend_;
	}
	bool getCmdHold(){
		return hold_;
	}
	bool getCmdUnhold(){
		return unhold_;
	}
	bool getCmdComplete(){
		return complete_;
	}
	bool getCmdStateComplete(){
		return stateComplete_;
	}

	void resetCmdAbort();
	void resetCmdStop();
	void resetCmdClear();
	void resetCmdReset();
	void resetCmdStart();
	void resetCmdSuspend();
	void resetCmdUnsuspend();
	void resetCmdHold();
	void resetCmdUnhold();
	void resetCmdComplete();
	void resetCmdStateComplete();

	// **********************************************************

	PackMLModuleStateEnu getParentCurrentState();

	long int getParentCurrentSubState();

	const char *getParentName();

	bool getParentStateComplete();

	PackMLModule* getParentAdr() { return pParentLink_; }

	bool getSiblingsStateComplete();

	bool getChildrenStateComplete();

	const char *getCurrentStateStr() const;

	const char *getStateStr(PackMLModuleStateEnu state) const;

	const char *getCurrentModeStr() const;

	unsigned long getChildCount() { return childCount_; }

	unsigned long getSiblingCount();

	unsigned short getHierarchyLevel()
	{
		return hierarchyLevel_;
	}

	// ************************* Service interface methods *********************
	// Name of the module
	const char* getModuleName() { return moduleName_.c_str(); }
	unsigned long int getModuleId() { return moduleId_; }

	// Called by the IEC function
	const char* getStateInfo() { return stateInfo_.c_str(); }

	bool setCurrentMode(long int mode);
	long int getCurrentMode(){ return modeCurrent_; }
	const char* getCurrentModeName() const;
	const char* getModeName(signed long int modeId) const;
	bool isModeChangePossible();

	bool getModuleReady() { return moduleReady_; }
	void setModuleReady(bool value);

	void setNewModeCurrent(long int mode);
	void setHierarchyLevel(unsigned short level);
	void setAllStateComplete();

	bool registerChild(PackMLModule* pChild); // called during onCreated()
	bool unregisterChild(PackMLModule* pChild);

	void escalateCmdAbort();
	void escalateCmdClear();

	void escalateCmdSuspend();
	void escalateCmdUnsuspend();

	void escalateCmdHold();
	void escalateCmdUnhold();

	void escalateCmdStop();
	void escalateCmdReset();

	void escalateCmdStart();
	void escalateCmdComplete();

	void propagateCmdAbort(bool root);
	void propagateCmdClear(bool root);

	void propagateCmdSuspend(bool root);
	void propagateCmdUnsuspend(bool root);

	void propagateCmdHold(bool root);
	void propagateCmdUnhold(bool root);

	void propagateCmdStop(bool root);
	void propagateCmdReset(bool root);

	void propagateCmdStart(bool root);
	void propagateCmdComplete(bool root);

	PackMLModuleStateEnu getCurrentState(){
		return stateCurrent_;
	}

	void setCurrentSubState(long int subState){
		subStateCurrent_ = subState;
		timeInSubState_ = 0.0;
	}

	long int getCurrentSubState(){
		return subStateCurrent_;
	}

	bool getStateComplete(){
		return stateComplete_;
	}
	// check if child wants to be synchronised
	bool needParentSynch(PackMLModuleStateEnu parentState);

	void setSharedInfoPtrs(PackMLModuleSharedInfo* pWaitingFor, PackMLModuleSharedInfo* pInteruptedBy);

	void setActivationPv(bool activationPv) { activationPv_ = activationPv; }

	PackMLModuleSharedInfo* getWaitingForPtr() {
		return pWaitingFor_;
	}

	PackMLModuleSharedInfo* getInteruptedByPtr() {
		return pInteruptedBy_;
	}

	PackMLModuleStateEnu getChildCurrentState(unsigned long int childIndex);
	long int getChildCurrentSubState(unsigned long int childIndex);
	bool getChildStateComplete(unsigned long int childIndex);
	const char* getChildName(unsigned long int childIndex);

	PackMLModuleStateEnu getSiblingCurrentState(unsigned long int siblingIndex);
	long int getSiblingCurrentSubState(unsigned long int siblingIndex);
	bool getSiblingStateComplete(unsigned long int siblingIndex);
	const char* getSiblingName(unsigned long int siblingIndex);

	float getTimeInState() { return timeInState_; }
	float getTimeInSubState() { return timeInSubState_; }

	void setCycleTime(float cycleTime) { cycleTime_ = cycleTime; }

	PackMLModule* getParentPtr();
	PackMLModule* getChildPtr(unsigned long int childIdx);
	PackMLModule* getSiblingPtr(unsigned long int siblingIdx);

	void* createUserMemory(unsigned long int userMemorySize);
	void* getUserMemoryPtr();
	void deleteUserMemory();

	bool isActingState(PackMLModuleStateEnu state);
	bool isWaitingState(PackMLModuleStateEnu state){
		return !isActingState(state);
	}

	void setInteruptedBy(PackMLModule* pPackMLModule);

	void setStateInfo(std::string stateInfo){
		stateInfo_ = stateInfo;
	}

	private:

	// --------------------------------------------------------
	// **************** Will be private ***********************
	// --------------------------------------------------------

	// unique service name identifier
	std::string moduleName_;
	unsigned long moduleId_;
	unsigned long generateId_(const char *pName);

	// used during the registration
	AtomicSemaphore semaphore_;

	// **************** FB parameters placeholder ******************
	std::string stateInfo_;

	short int activationCondition_;

	bool overrideAbort_;
	bool overrideStop_;
	bool overrideClear_;
	bool overrideReset_;
	bool overrideStart_;
	bool overrideSuspend_;
	bool overrideUnsuspend_;
	bool overrideHold_;
	bool overrideUnhold_;
	bool overrideComplete_;

	bool reactToAbort_;
	bool reactToStop_;
	bool reactToClear_;
	bool reactToReset_;
	bool reactToStart_;
	bool reactToSuspend_;
	bool reactToUnsuspend_;
	bool reactToHold_;
	bool reactToUnhold_;
	bool reactToComplete_;

	bool escalateAbort_;
	bool escalateStop_;
	bool escalateClear_;
	bool escalateReset_;
	bool escalateStart_;
	bool escalateSuspend_;
	bool escalateUnsuspend_;
	bool escalateHold_;
	bool escalateUnhold_;
	bool escalateComplete_;

	// ****************** Hierarchy related stuff ***********************

	// Pointers to the parent/childs in the hierarchy
	// Change it to smart pointers
	PackMLModule* pParentLink_;
	std::vector<PackMLModule*> childLinks_;
	unsigned long int parentLinkAdr_;

	// Configure the hierarchy
	bool linkToParent_(PackMLModule* pParent);
	bool unlinkFromParent_();

	bool hasParent_;
	unsigned long childCount_;
	unsigned short hierarchyLevel_;

	bool moduleReady_;

	// *************** PackML State Manager *******************
	long int modeCurrent_;
	PackMLModuleStateEnu stateCurrent_;
	long int subStateCurrent_;

	bool activate_;
	bool deactivate_;

	// Internal cmds
	bool abort_;
	bool clear_;
	bool stop_;
	bool reset_;
	bool start_;
	bool hold_;
	bool unhold_;
	bool suspend_;
	bool unsuspend_;
	bool complete_;
	bool stateComplete_;

	bool oldAbort_;
	bool oldClear_;
	bool oldStop_;
	bool oldReset_;
	bool oldStart_;
	bool oldHold_;
	bool oldUnhold_;
	bool oldSuspend_;
	bool oldUnsuspend_;
	bool oldComplete_;
	bool oldStateComplete_;

	bool externalAbort_;
	bool externalClear_;
	bool externalStop_;
	bool externalReset_;
	bool externalStart_;
	bool externalHold_;
	bool externalUnhold_;
	bool externalSuspend_;
	bool externalUnsuspend_;
	bool externalComplete_;
	bool externalStateComplete_;

	void updatePackMLModel_();

	void checkActivationCondition_();

	void checkParentStateCondition_();

	bool setCmd_(PackMLModuleStateEnu targetActingState);
	void resetCmd_(PackMLModuleStateEnu targetActingState);

	void executeCmd_(PackMLModuleStateEnu targetState);

	void executeActingState_(PackMLModuleStateEnu targetState);

	bool stateExistInPattern_(unsigned long stateBitPattern,
	PackMLModuleStateEnu state);

	bool cmdValid_(PackMLModuleStateEnu state);
	// Checks if the all the children are in the provided state
	bool childrenInState_(PackMLModuleStateEnu state);
	// Checks if the children are in need of synchronisation for the provided
	// state
	bool childrenInSynch_(PackMLModuleStateEnu targetState);

	bool isChild_(PackMLModule* pModule);

	// Reset the cmds, substate, status etc when a state changes
	void resetInternalCmds_();

	// Waiting for and aborted by related stuff
	void setWaitingFor_();
	void resetWaitingFor_();
	void setInteruptedBy_();
	void resetInteruptedBy_();

	PackMLModuleSharedInfo* pWaitingFor_;
	PackMLModuleSharedInfo* pInteruptedBy_;

	bool activationPv_;
	float timeInState_;
	float timeInSubState_;
	float cycleTime_; // ms

	void updateTimeInState_() {
		timeInState_ += cycleTime_;
		timeInSubState_ += cycleTime_;
	}

	void* pUserData_;
	unsigned long int userDataSize_;

};

#endif // __MAPP_MXPACKML_PACKMLMODULE_HPP__
```

#### PackMLModule.cpp
```cpp
#include "PackMLModule.hpp"

		// -----------------------------------------------------------------------------

PackMLModule::PackMLModule(const char* pModuleName) : moduleName_(pModuleName),
	moduleId_(0),
	semaphore_(),
	activationCondition_(0),
	overrideAbort_(false),
	overrideStop_(false),
	overrideClear_(false),
	overrideReset_(false),
	overrideStart_(false),
	overrideSuspend_(false),
	overrideUnsuspend_(false),
	overrideHold_(false),
	overrideUnhold_(false),
	overrideComplete_(false),
	reactToAbort_(false),
	reactToStop_(false),
	reactToClear_(false),
	reactToReset_(false),
	reactToStart_(false),
	reactToSuspend_(false),
	reactToUnsuspend_(false),
	reactToHold_(false),
	reactToUnhold_(false),
	reactToComplete_(false),
	escalateAbort_(false),
	escalateStop_(false),
	escalateClear_(false),
	escalateReset_(false),
	escalateStart_(false),
	escalateSuspend_(false),
	escalateUnsuspend_(false),
	escalateHold_(false),
	escalateUnhold_(false),
	escalateComplete_(false),
	pParentLink_(nullptr),
	childLinks_(),
	parentLinkAdr_(0),
	hasParent_(false),
	childCount_(0),
	hierarchyLevel_(0),
	moduleReady_(false),
	modeCurrent_(1),
	stateCurrent_(ST_UNDEFINED),
	subStateCurrent_(0),
	activate_(false),
	deactivate_(false),
	abort_(false),
	clear_(false),
	stop_(false),
	reset_(false),
	start_(false),
	hold_(false),
	unhold_(false),
	suspend_(false),
	unsuspend_(false),
	complete_(false),
	stateComplete_(false),
	oldAbort_(false),
	oldClear_(false),
	oldStop_(false),
	oldReset_(false),
	oldStart_(false),
	oldHold_(false),
	oldUnhold_(false),
	oldSuspend_(false),
	oldUnsuspend_(false),
	oldComplete_(false),
	oldStateComplete_(false),
	externalAbort_(false),
	externalClear_(false),
	externalStop_(false),
	externalReset_(false),
	externalStart_(false),
	externalHold_(false),
	externalUnhold_(false),
	externalSuspend_(false),
	externalUnsuspend_(false),
	externalComplete_(false),
	externalStateComplete_(false),
	pWaitingFor_(nullptr),
	pInteruptedBy_(nullptr),
	activationPv_(false),
	timeInState_(0.0),
	timeInSubState_(0.0),
	cycleTime_(0.0),
	pUserData_(nullptr),
	userDataSize_(0)
{
	//	moduleName_ = "";
	stateInfo_ = "";
	moduleId_ = generateId_(pModuleName);

}

		// -----------------------------------------------------------------------------

PackMLModule::~PackMLModule()
{
	free(pUserData_);
}

// -----------------------------------------------------------------------------
void* PackMLModule::createUserMemory(unsigned long int userMemorySize){
	if(pUserData_ != nullptr)
		return pUserData_;

	pUserData_ = calloc(userMemorySize, sizeof(char));
	userDataSize_ = userMemorySize;
//	memset(pUserData_, 0, userDataSize_);

	return pUserData_;
}
// -----------------------------------------------------------------------------
void* PackMLModule::getUserMemoryPtr(){
	return pUserData_;
}

void PackMLModule::deleteUserMemory(){
	free(pUserData_);
}

// -----------------------------------------------------------------------------

void PackMLModule::initModule()
{
	setNewModeCurrent(modeCurrent_);
	setHierarchyLevel(0);

	if(pWaitingFor_ == nullptr)
		pWaitingFor_ = new PackMLModuleSharedInfo();
	if(pInteruptedBy_ == nullptr)
		pInteruptedBy_ = new PackMLModuleSharedInfo();

	setSharedInfoPtrs(pWaitingFor_, pInteruptedBy_);
	setModuleReady(true);

}

bool PackMLModule::initModule(PackMLModule* pParent)
{
	if(pParent == nullptr || pParent == this || isChild_(pParent)){
		return false;
	}
	return linkToParent_(pParent);
}

		// -----------------------------------------------------------------------------
bool PackMLModule::exitModule()
{
	// decide what to do here, do we need to reset those when unlinking from parent
	resetWaitingFor_();
	resetInteruptedBy_();

	// ******
	// nested call for resetWaitingFor and InteruptedBy for all children and childrens children
	// ******

	setNewModeCurrent(modeCurrent_);
	setHierarchyLevel(0);
	setModuleReady(false);

	stateInfo_ = "";

	overrideAbort_ = false;
	overrideStop_ = false;
	overrideClear_ = false;
	overrideReset_ = false;
	overrideStart_ = false;
	overrideSuspend_ = false;
	overrideUnsuspend_ = false;
	overrideHold_ = false;
	overrideUnhold_ = false;
	overrideComplete_ = false;
	reactToAbort_ = false;
	reactToStop_ = false;
	reactToClear_ = false;
	reactToReset_ = false;
	reactToStart_ = false;
	reactToSuspend_ = false;
	reactToUnsuspend_ = false;
	reactToHold_ = false;
	reactToUnhold_ = false;
	reactToComplete_ = false;
	escalateAbort_ = false;
	escalateStop_ = false;
	escalateClear_ = false;
	escalateReset_ = false;
	escalateStart_ = false;
	escalateSuspend_ = false;
	escalateUnsuspend_ = false;
	escalateHold_ = false;
	escalateUnhold_ = false;
	escalateComplete_ = false;
	activate_ = false;
	deactivate_ = false;

	resetInternalCmds_();

	if(!hasParent_){
		delete pWaitingFor_;
		delete pInteruptedBy_;
		setSharedInfoPtrs(nullptr, nullptr);
		return true;
	}

	setSharedInfoPtrs(nullptr, nullptr);
	return unlinkFromParent_();
}

		// -----------------------------------------------------------------------------

void PackMLModule::runPackMLModule()
{
	updateTimeInState_();
	// check parent state condition
	checkParentStateCondition_();
	// update the packml model
	updatePackMLModel_();

}
		// ---------------------------------------------------------------------------

		// called during onCreated() if parent found and in onService()
bool PackMLModule::linkToParent_(PackMLModule* pParent)
{
	if(pParent->registerChild(this)){
		pParentLink_ = pParent;
		hasParent_ = true;
		return true;
	}
	return false;
}

		// -------------------------------------------------------------------------

bool PackMLModule::unlinkFromParent_()
{
	if(pParentLink_->unregisterChild(this)){
		pParentLink_ = nullptr;
		hasParent_ = false;
		return true;
	}
	return false;
}

		// -------------------------------------------------------------------------

bool PackMLModule::registerChild(PackMLModule* pChild)
{

	if(isChild_(pChild))
		return true;

	if(!semaphore_.acquire())
		return false;

	childLinks_.push_back(pChild);

	pChild->setNewModeCurrent(modeCurrent_);
	pChild->setHierarchyLevel(hierarchyLevel_ + 1);
	pChild->setSharedInfoPtrs(pWaitingFor_, pInteruptedBy_);
	pChild->setModuleReady(moduleReady_);

	childCount_ = childLinks_.size();
	semaphore_.release();
	return true;
}

		// -------------------------------------------------------------------------

bool PackMLModule::unregisterChild(PackMLModule* pChild)
{
	//			BR::Core::MutexLocker lock(&mutex_);

	if(!semaphore_.acquire())
		return false;

	for (unsigned short i = 0; i < childCount_; ++i) {
		if (childLinks_[i]->getModuleId() == pChild->getModuleId()) {
			childLinks_.erase(childLinks_.begin() + i);
			break;
		}
	}

	childCount_ = childLinks_.size();
	semaphore_.release();
	return true;
}

		// -------------------------------------------------------------------------

void PackMLModule::setModuleReady(bool value)
{
	moduleReady_ = value;

	if (moduleReady_) {
		stateCurrent_ = ST_DEACTIVATED;
	}
	else {
		stateCurrent_ = ST_UNDEFINED;
	}

	for (unsigned short i = 0; i < childCount_; ++i) {
		childLinks_[i]->setModuleReady(value);
	}
}

void PackMLModule::setHierarchyLevel(unsigned short level)
{
	hierarchyLevel_ = level;

	for (unsigned short i = 0; i < childCount_; ++i) {
		childLinks_[i]->setHierarchyLevel(level + 1);
	}

}

void PackMLModule::setAllStateComplete()
{
	stateComplete_ = true;
	externalStateComplete_ = stateComplete_;

	for (unsigned short i = 0; i < childCount_; ++i) {
		childLinks_[i]->setAllStateComplete();
	}

}

void PackMLModule::setSharedInfoPtrs(PackMLModuleSharedInfo* pWaitingFor, PackMLModuleSharedInfo* pInteruptedBy)
{
	pWaitingFor_ = pWaitingFor;
	pInteruptedBy_ = pInteruptedBy;

	for (unsigned short i = 0; i < childCount_; ++i) {
		childLinks_[i]->setSharedInfoPtrs(pWaitingFor_, pInteruptedBy_);
	}

}

		// -------------------------------------------------------------------------

unsigned long PackMLModule::generateId_(const char *pName)
{
	unsigned long int N = strlen(pName);
	unsigned long int b    = 378551;
	unsigned long int a    = 63689;
	unsigned long int hash = 0;

	for(std::size_t i = 0; i < N; i++)
	{
		hash = hash * a + pName[i];
		a    = a * b;
	}

	return (hash & 0x7FFFFFFF);
}
```
